C07303=1117.265,17.086,-52.064,179.768,6.707,149.300
C07304=1117.260,17.335,-52.079,179.769,6.711,149.301
C07305=1117.255,17.584,-52.094,179.769,6.716,149.302
C07306=1117.250,17.834,-52.108,179.770,6.720,149.303
C07307=1117.245,18.084,-52.123,179.771,6.725,149.303
C07308=1117.240,18.333,-52.138,179.772,6.729,149.304
C07309=1117.235,18.583,-52.152,179.773,6.734,149.305
C07310=1117.230,18.832,-52.168,179.774,6.738,149.306
C07311=1117.225,19.082,-52.182,179.774,6.742,149.306
C07312=1117.220,19.332,-52.196,179.775,6.747,149.307
C07313=1117.215,19.581,-52.211,179.776,6.751,149.308
C07314=1117.210,19.831,-52.226,179.776,6.756,149.309
C07315=1117.205,20.080,-52.241,179.777,6.760,149.309
C07316=1117.200,20.330,-52.255,179.778,6.764,149.310
C07317=1117.195,20.579,-52.271,179.779,6.769,149.311
C07318=1117.190,20.829,-52.285,179.780,6.773,149.312
C07319=1117.185,21.078,-52.300,179.781,6.778,149.312
C07320=1117.179,21.328,-52.315,179.782,6.782,149.313
C07321=1117.175,21.577,-52.330,179.783,6.787,149.314
C07322=1117.170,21.827,-52.344,179.783,6.791,149.315
C07323=1117.164,22.076,-52.360,179.784,6.796,149.315
C07324=1117.160,22.291,-52.372,179.785,6.799,149.316
C07325=1117.155,22.505,-52.385,179.785,6.803,149.317
C07326=1117.151,22.720,-52.397,179.786,6.807,149.317
C07327=1117.147,22.935,-52.410,179.787,6.810,149.318
C07328=1117.142,23.149,-52.424,179.787,6.814,149.318
C07329=1117.139,23.364,-52.436,179.788,6.818,149.319
C07330=1117.134,23.579,-52.449,179.789,6.822,149.320
C07331=1117.130,23.793,-52.462,179.790,6.826,149.320
C07332=1117.125,24.043,-52.477,179.790,6.829,149.321
C07333=1117.120,24.292,-52.492,179.791,6.834,149.322
C07334=1117.114,24.542,-52.507,179.792,6.838,149.322
C07335=1117.110,24.791,-52.522,179.793,6.843,149.323
C07336=1117.105,25.041,-52.537,179.794,6.847,149.324
C07337=1117.099,25.290,-52.552,179.795,6.851,149.324
C07338=1117.095,25.539,-52.567,179.796,6.856,149.325
C07339=1117.089,25.789,-52.582,179.797,6.860,149.326
C07340=1117.084,26.038,-52.597,179.798,6.865,149.327
C07341=1117.079,26.288,-52.613,179.799,6.869,149.327
C07342=1117.074,26.537,-52.628,179.800,6.873,149.328
C07343=1117.069,26.787,-52.643,179.800,6.877,149.329
C07344=1117.065,27.036,-52.658,179.801,6.882,149.329
C07345=1117.059,27.286,-52.673,179.802,6.886,149.330
C07346=1117.054,27.536,-52.688,179.803,6.890,149.331
C07347=1117.049,27.785,-52.703,179.804,6.895,149.331
C07348=1117.044,28.034,-52.718,179.805,6.899,149.332
C07349=1117.039,28.283,-52.734,179.806,6.904,149.333
C07350=1117.034,28.533,-52.749,179.807,6.908,149.334
C07351=1117.029,28.783,-52.764,179.808,6.912,149.334
C07352=1117.025,29.032,-52.779,179.809,6.917,149.335
C07353=1117.019,29.282,-52.795,179.809,6.920,149.336
C07354=1117.014,29.531,-52.810,179.810,6.924,149.336
C07355=1117.009,29.780,-52.825,179.812,6.929,149.337
C07356=1117.004,30.030,-52.841,179.813,6.933,149.337
C07357=1116.999,30.280,-52.855,179.814,6.937,149.338
C07358=1116.994,30.529,-52.871,179.815,6.942,149.339
C07359=1116.989,30.779,-52.886,179.815,6.946,149.340
C07360=1116.984,31.028,-52.902,179.816,6.951,149.340
C07361=1116.979,31.277,-52.917,179.817,6.955,149.341
C07362=1116.974,31.527,-52.933,179.818,6.958,149.342
C07363=1116.969,31.777,-52.948,179.819,6.963,149.342
C07364=1116.964,32.026,-52.963,179.820,6.967,149.343
C07365=1116.959,32.275,-52.979,179.821,6.971,149.344
C07366=1116.954,32.524,-52.994,179.822,6.976,149.344
C07367=1116.950,32.774,-53.010,179.823,6.980,149.345
C07368=1116.944,33.024,-53.025,179.824,6.984,149.346
C07369=1116.939,33.273,-53.041,179.825,6.989,149.346
C07370=1116.934,33.522,-53.056,179.826,6.993,149.347
C07371=1116.929,33.772,-53.072,179.827,6.996,149.347
C07372=1116.924,34.022,-53.087,179.828,7.001,149.348
C07373=1116.919,34.271,-53.102,179.829,7.005,149.349
C07374=1116.914,34.520,-53.118,179.830,7.009,149.349
C07375=1116.909,34.770,-53.134,179.831,7.014,149.350
C07376=1116.905,35.019,-53.149,179.832,7.018,149.351
C07377=1116.899,35.269,-53.164,179.833,7.022,149.351
C07378=1116.894,35.518,-53.180,179.834,7.027,149.352
C07379=1116.889,35.768,-53.196,179.835,7.031,149.353
C07380=1116.885,35.983,-53.210,179.836,7.034,149.353
C07381=1116.881,36.197,-53.222,179.837,7.038,149.354
C07382=1116.877,36.412,-53.236,179.838,7.041,149.354
C07383=1116.872,36.626,-53.250,179.839,7.045,149.355
C07384=1116.868,36.841,-53.263,179.840,7.048,149.355
C07385=1116.863,37.055,-53.276,179.841,7.052,149.356
C07386=1116.859,37.269,-53.290,179.842,7.056,149.356
C07387=1116.855,37.484,-53.304,179.842,7.059,149.357
C07388=1116.849,37.733,-53.319,179.843,7.063,149.358
C07389=1116.845,37.983,-53.335,179.845,7.067,149.358
C07390=1116.840,38.232,-53.350,179.846,7.072,149.359
C07391=1116.835,38.482,-53.366,179.847,7.076,149.359
C07392=1116.830,38.732,-53.382,179.848,7.080,149.360
C07393=1116.825,38.981,-53.398,179.848,7.084,149.361
C07394=1116.819,39.230,-53.414,179.849,7.088,149.361
C07395=1116.815,39.480,-53.430,179.850,7.092,149.362
C07396=1116.810,39.729,-53.445,179.852,7.096,149.362
C07397=1116.805,39.978,-53.461,179.853,7.101,149.363
C07398=1116.800,40.228,-53.477,179.854,7.105,149.364
C07399=1116.795,40.478,-53.492,179.855,7.109,149.364
C07400=1116.789,40.727,-53.508,179.856,7.114,149.365
C07401=1116.785,40.976,-53.525,179.857,7.117,149.366
C07402=1116.779,41.226,-53.540,179.858,7.121,149.366
C07403=1116.775,41.476,-53.556,179.859,7.125,149.367
C07404=1116.770,41.724,-53.572,179.860,7.130,149.367
C07405=1116.765,41.974,-53.588,179.861,7.134,149.368
C07406=1116.760,42.224,-53.603,179.863,7.138,149.369
C07407=1116.755,42.473,-53.620,179.864,7.142,149.369
C07408=1116.750,42.723,-53.636,179.865,7.146,149.370
C07409=1116.745,42.972,-53.651,179.866,7.150,149.370
C07410=1116.740,43.221,-53.668,179.867,7.154,149.371
C07411=1116.735,43.471,-53.684,179.868,7.158,149.372
C07412=1116.730,43.720,-53.700,179.869,7.162,149.372
C07413=1116.725,43.970,-53.716,179.870,7.167,149.373
C07414=1116.720,44.219,-53.731,179.871,7.171,149.374
C07415=1116.715,44.469,-53.748,179.873,7.175,149.374
C07416=1116.710,44.718,-53.764,179.873,7.178,149.375
C07417=1116.705,44.967,-53.780,179.875,7.183,149.375
C07418=1116.700,45.217,-53.796,179.876,7.187,149.376
C07419=1116.695,45.466,-53.812,179.877,7.191,149.376
C07420=1116.690,45.716,-53.828,179.878,7.195,149.377
C07421=1116.685,45.965,-53.844,179.879,7.200,149.378
C07422=1116.680,46.215,-53.860,179.881,7.204,149.378
C07423=1116.675,46.464,-53.877,179.882,7.208,149.379
C07424=1116.670,46.714,-53.893,179.882,7.211,149.379
C07425=1116.665,46.963,-53.909,179.884,7.215,149.380
C07426=1116.660,47.213,-53.925,179.885,7.220,149.380
C07427=1116.655,47.461,-53.941,179.886,7.224,149.381
C07428=1116.651,47.711,-53.958,179.888,7.228,149.382
C07429=1116.646,47.960,-53.974,179.889,7.232,149.382
C07430=1116.641,48.210,-53.990,179.890,7.236,149.383
C07431=1116.636,48.459,-54.006,179.891,7.240,149.383
C07432=1116.631,48.709,-54.022,179.892,7.244,149.384
C07433=1116.626,48.958,-54.039,179.893,7.248,149.384
C07434=1116.621,49.208,-54.055,179.895,7.252,149.385
C07435=1116.616,49.457,-54.072,179.896,7.256,149.386
C07436=1116.610,49.781,-54.093,179.897,7.261,149.386
C07437=1116.603,50.104,-54.114,179.899,7.267,149.387
C07438=1116.597,50.427,-54.135,179.900,7.272,149.388
C07439=1116.591,50.750,-54.156,179.902,7.277,149.388
C07440=1116.585,51.000,-54.173,179.903,7.281,149.389
C07441=1116.580,51.249,-54.190,179.905,7.285,149.390
C07442=1116.576,51.499,-54.206,179.906,7.290,149.390
C07443=1116.571,51.748,-54.222,179.906,7.293,149.391
C07444=1116.566,51.997,-54.239,179.908,7.297,149.391
C07445=1116.560,52.247,-54.255,179.909,7.301,149.392
C07446=1116.556,52.497,-54.271,179.910,7.305,149.392
C07447=1116.550,52.745,-54.288,179.911,7.309,149.393
C07448=1116.546,52.995,-54.304,179.913,7.313,149.393
C07449=1116.541,53.245,-54.322,179.914,7.318,149.394
C07450=1116.536,53.493,-54.338,179.915,7.322,149.395
C07451=1116.531,53.744,-54.354,179.916,7.325,149.395
C07452=1116.526,53.993,-54.371,179.917,7.329,149.396
C07453=1116.521,54.242,-54.387,179.919,7.333,149.396
C07454=1116.516,54.492,-54.404,179.920,7.338,149.397
C07455=1116.511,54.740,-54.420,179.921,7.342,149.397
C07456=1116.507,54.990,-54.437,179.923,7.346,149.398
C07457=1116.501,55.240,-54.454,179.924,7.350,149.398
C07458=1116.496,55.489,-54.470,179.925,7.354,149.399
C07459=1116.491,55.739,-54.487,179.926,7.357,149.399
C07460=1116.486,55.988,-54.504,179.927,7.361,149.400
C07461=1116.481,56.237,-54.520,179.929,7.365,149.401
C07462=1116.477,56.487,-54.537,179.930,7.370,149.401
C07463=1116.471,56.736,-54.554,179.931,7.374,149.402
C07464=1116.465,57.091,-54.578,179.933,7.379,149.402
C07465=1116.458,57.446,-54.601,179.935,7.385,149.403
C07466=1116.450,57.801,-54.626,179.937,7.391,149.404
C07467=1116.444,58.155,-54.649,179.939,7.396,149.405
C07468=1116.438,58.405,-54.666,179.940,7.401,149.405
C07469=1116.434,58.655,-54.683,179.941,7.404,149.406
C07470=1116.429,58.903,-54.699,179.942,7.409,149.406
C07471=1116.424,59.153,-54.716,179.944,7.413,149.407
C07472=1116.419,59.403,-54.733,179.944,7.416,149.407
C07473=1116.414,59.652,-54.750,179.946,7.420,149.408
C07474=1116.409,59.901,-54.767,179.947,7.424,149.409
C07475=1116.404,60.151,-54.784,179.949,7.428,149.409
C07476=1116.399,60.400,-54.801,179.950,7.432,149.409
C07477=1116.394,60.649,-54.818,179.951,7.436,149.410
C07478=1116.389,60.898,-54.835,179.953,7.440,149.410
C07479=1116.385,61.148,-54.852,179.954,7.445,149.411
C07480=1116.379,61.398,-54.869,179.955,7.449,149.412
C07481=1116.375,61.647,-54.886,179.956,7.452,149.412
C07482=1116.369,61.896,-54.902,179.958,7.456,149.413
C07483=1116.365,62.145,-54.920,179.959,7.460,149.413
C07484=1116.360,62.395,-54.937,179.960,7.464,149.414
C07485=1116.355,62.644,-54.954,179.962,7.468,149.414
C07486=1116.350,62.894,-54.971,179.963,7.472,149.415
C07487=1116.345,63.143,-54.987,179.964,7.476,149.415
C07488=1116.341,63.358,-55.003,179.965,7.479,149.416
C07489=1116.337,63.571,-55.017,179.966,7.483,149.416
C07490=1116.333,63.786,-55.033,179.968,7.486,149.417
C07491=1116.328,64.001,-55.046,179.969,7.490,149.417
C07492=1116.324,64.215,-55.061,179.970,7.493,149.417
C07493=1116.320,64.429,-55.076,179.971,7.497,149.418
C07494=1116.316,64.643,-55.091,179.972,7.500,149.418
C07495=1116.311,64.858,-55.106,179.974,7.504,149.419
C07496=1116.307,65.107,-55.123,179.974,7.507,149.419
C07497=1116.301,65.356,-55.140,179.976,7.511,149.420
C07498=1116.297,65.606,-55.157,179.977,7.515,149.420
C07499=1116.292,65.855,-55.175,179.979,7.519,149.421
C07500=1116.287,66.104,-55.191,179.980,7.523,149.421
C07501=1116.282,66.354,-55.209,179.982,7.527,149.422
C07502=1116.277,66.603,-55.227,179.983,7.531,149.422
C07503=1116.273,66.853,-55.243,179.984,7.535,149.423
C07504=1116.267,67.102,-55.260,179.986,7.540,149.423
C07505=1116.262,67.351,-55.278,179.987,7.543,149.424
C07506=1116.258,67.601,-55.295,179.988,7.547,149.424
C07507=1116.253,67.850,-55.313,179.989,7.551,149.425
C07508=1116.247,68.100,-55.330,179.991,7.555,149.425
C07509=1116.243,68.348,-55.347,179.992,7.559,149.426
C07510=1116.238,68.598,-55.365,179.993,7.563,149.426
C07511=1116.233,68.847,-55.383,179.995,7.567,149.427
C07512=1116.229,69.097,-55.399,179.997,7.571,149.427
C07513=1116.224,69.346,-55.417,179.998,7.575,149.428
C07514=1116.218,69.596,-55.435,179.999,7.579,149.428
C07515=1116.214,69.844,-55.452,-179.999,7.583,149.429
C07516=1116.208,70.094,-55.469,-179.998,7.587,149.429
C07517=1116.204,70.343,-55.487,-179.997,7.590,149.430
C07518=1116.198,70.593,-55.504,-179.996,7.594,149.430
C07519=1116.194,70.842,-55.521,-179.994,7.598,149.431
C07520=1116.189,71.091,-55.539,-179.993,7.602,149.431
C07521=1116.184,71.341,-55.557,-179.991,7.606,149.432
C07522=1116.179,71.590,-55.574,-179.990,7.610,149.432
C07523=1116.175,71.839,-55.591,-179.989,7.614,149.433
C07524=1116.170,72.088,-55.609,-179.987,7.618,149.433
C07525=1116.165,72.338,-55.627,-179.985,7.622,149.434
C07526=1116.160,72.587,-55.645,-179.984,7.626,149.434
C07527=1116.155,72.837,-55.663,-179.983,7.630,149.435
C07528=1116.150,73.086,-55.679,-179.981,7.634,149.435
C07529=1116.145,73.335,-55.697,-179.980,7.638,149.436
C07530=1116.140,73.585,-55.714,-179.979,7.642,149.436
C07531=1116.135,73.834,-55.732,-179.978,7.646,149.437
C07532=1116.130,74.083,-55.750,-179.976,7.650,149.437
C07533=1116.125,74.333,-55.768,-179.974,7.653,149.438
C07534=1116.121,74.582,-55.785,-179.973,7.658,149.438
C07535=1116.116,74.831,-55.803,-179.972,7.662,149.439
C07536=1116.111,75.080,-55.821,-179.970,7.666,149.439
C07537=1116.106,75.330,-55.839,-179.969,7.669,149.440
C07538=1116.101,75.579,-55.856,-179.967,7.674,149.440
C07539=1116.096,75.829,-55.874,-179.966,7.678,149.441
C07540=1116.091,76.078,-55.892,-179.964,7.681,149.441
C07541=1116.086,76.327,-55.910,-179.963,7.685,149.442
C07542=1116.082,76.577,-55.928,-179.962,7.690,149.442
C07543=1116.077,76.827,-55.946,-179.960,7.694,149.443
C07544=1116.073,77.040,-55.961,-179.959,7.697,149.443
C07545=1116.069,77.254,-55.976,-179.958,7.700,149.444
C07546=1116.064,77.468,-55.991,-179.958,7.703,149.444
C07547=1116.060,77.683,-56.007,-179.957,7.706,149.445
C07548=1116.056,77.897,-56.023,-179.956,7.709,149.445
C07549=1116.051,78.111,-56.038,-179.955,7.712,149.445
C07550=1116.047,78.326,-56.053,-179.954,7.715,149.446
C07551=1116.043,78.541,-56.069,-179.954,7.718,149.447
C07552=1116.038,78.790,-56.087,-179.952,7.722,149.447
C07553=1116.033,79.039,-56.105,-179.952,7.726,149.448
C07554=1116.028,79.288,-56.123,-179.950,7.730,149.448
C07555=1116.024,79.537,-56.141,-179.950,7.733,149.449
C07556=1116.019,79.787,-56.159,-179.948,7.737,149.449
C07557=1116.014,80.036,-56.177,-179.948,7.741,149.450
C07558=1116.009,80.285,-56.195,-179.946,7.745,149.450
C07559=1116.004,80.534,-56.213,-179.945,7.748,149.451
C07560=1116.000,80.784,-56.231,-179.944,7.752,149.451
C07561=1115.995,81.033,-56.249,-179.943,7.756,149.452
C07562=1115.990,81.282,-56.267,-179.942,7.760,149.453
C07563=1115.985,81.532,-56.285,-179.941,7.764,149.453
C07564=1115.980,81.781,-56.303,-179.940,7.767,149.453
C07565=1115.975,82.030,-56.321,-179.939,7.771,149.454
C07566=1115.971,82.280,-56.339,-179.938,7.774,149.454
C07567=1115.966,82.529,-56.357,-179.936,7.778,149.455
C07568=1115.961,82.778,-56.375,-179.935,7.782,149.456
C07569=1115.956,83.027,-56.393,-179.934,7.786,149.456
C07570=1115.951,83.276,-56.411,-179.933,7.790,149.457
C07571=1115.946,83.526,-56.429,-179.932,7.794,149.457
C07572=1115.942,83.776,-56.447,-179.931,7.797,149.458
C07573=1115.936,84.025,-56.466,-179.930,7.801,149.458
C07574=1115.931,84.274,-56.484,-179.929,7.804,149.459
C07575=1115.926,84.523,-56.502,-179.927,7.808,149.459
C07576=1115.922,84.772,-56.521,-179.926,7.813,149.460
C07577=1115.917,85.022,-56.539,-179.925,7.816,149.460
C07578=1115.913,85.271,-56.557,-179.924,7.820,149.461
C07579=1115.908,85.520,-56.575,-179.922,7.824,149.461
C07580=1115.902,85.770,-56.593,-179.921,7.827,149.462
C07581=1115.898,86.020,-56.612,-179.920,7.831,149.462
C07582=1115.893,86.269,-56.630,-179.919,7.835,149.463
C07583=1115.888,86.517,-56.648,-179.917,7.840,149.464
C07584=1115.883,86.766,-56.666,-179.916,7.843,149.464
C07585=1115.878,87.016,-56.684,-179.915,7.847,149.464
C07586=1115.873,87.266,-56.703,-179.914,7.851,149.465
C07587=1115.869,87.514,-56.722,-179.913,7.854,149.465
C07588=1115.864,87.764,-56.740,-179.911,7.858,149.466
C07589=1115.859,88.013,-56.758,-179.910,7.862,149.467
C07590=1115.854,88.263,-56.777,-179.908,7.866,149.467
C07591=1115.849,88.511,-56.796,-179.907,7.870,149.467
C07592=1115.844,88.761,-56.814,-179.906,7.873,149.468
C07593=1115.840,89.010,-56.832,-179.905,7.877,149.469
C07594=1115.834,89.260,-56.851,-179.903,7.881,149.469
C07595=1115.830,89.509,-56.869,-179.901,7.885,149.469
C07596=1115.825,89.758,-56.887,-179.901,7.888,149.470
C07597=1115.820,90.008,-56.906,-179.899,7.892,149.470
C07598=1115.815,90.256,-56.925,-179.898,7.896,149.471
C07599=1115.810,90.506,-56.943,-179.896,7.900,149.471
C07600=1115.806,90.720,-56.959,-179.895,7.903,149.472
C07601=1115.803,90.934,-56.975,-179.894,7.906,149.472
C07602=1115.798,91.149,-56.990,-179.893,7.910,149.473
C07603=1115.794,91.363,-57.007,-179.892,7.913,149.473
C07604=1115.789,91.576,-57.023,-179.891,7.917,149.473
C07605=1115.786,91.790,-57.039,-179.889,7.920,149.474
C07606=1115.782,92.005,-57.055,-179.888,7.923,149.474
C07607=1115.778,92.219,-57.070,-179.887,7.926,149.475
C07608=1115.772,92.468,-57.090,-179.885,7.930,149.475
C07609=1115.767,92.717,-57.108,-179.884,7.934,149.475
C07610=1115.763,92.967,-57.127,-179.882,7.938,149.476
C07611=1115.758,93.216,-57.145,-179.881,7.942,149.476
C07612=1115.754,93.465,-57.164,-179.879,7.946,149.477
C07613=1115.748,93.715,-57.183,-179.878,7.950,149.477
C07614=1115.744,93.963,-57.202,-179.877,7.953,149.478
C07615=1115.738,94.214,-57.221,-179.875,7.957,149.478
C07616=1115.734,94.462,-57.239,-179.873,7.961,149.479
C07617=1115.729,94.711,-57.257,-179.872,7.965,149.479
C07618=1115.724,94.961,-57.277,-179.870,7.969,149.480
C07619=1115.719,95.210,-57.295,-179.869,7.973,149.480
C07620=1115.715,95.460,-57.315,-179.867,7.976,149.480
C07621=1115.710,95.708,-57.333,-179.865,7.980,149.481
C07622=1115.705,95.958,-57.352,-179.864,7.984,149.481
C07623=1115.700,96.207,-57.371,-179.862,7.988,149.482
C07624=1115.695,96.456,-57.390,-179.861,7.992,149.482
C07625=1115.691,96.706,-57.409,-179.859,7.996,149.483
C07626=1115.685,96.954,-57.428,-179.857,8.000,149.483
C07627=1115.681,97.204,-57.446,-179.856,8.004,149.483
C07628=1115.676,97.453,-57.465,-179.854,8.008,149.484
C07629=1115.672,97.703,-57.485,-179.853,8.011,149.484
C07630=1115.666,97.952,-57.503,-179.851,8.015,149.485
C07631=1115.662,98.201,-57.522,-179.849,8.019,149.485
C07632=1115.657,98.450,-57.541,-179.847,8.023,149.485
C07633=1115.652,98.699,-57.559,-179.846,8.027,149.486
C07634=1115.647,98.949,-57.579,-179.844,8.030,149.486
C07635=1115.642,99.197,-57.598,-179.843,8.034,149.487
C07636=1115.638,99.447,-57.617,-179.841,8.038,149.487
C07637=1115.633,99.696,-57.635,-179.839,8.042,149.487
C07638=1115.628,99.946,-57.655,-179.837,8.046,149.488
C07639=1115.623,100.195,-57.674,-179.836,8.050,149.488
C07640=1115.619,100.444,-57.693,-179.834,8.053,149.489
C07641=1115.613,100.693,-57.713,-179.832,8.057,149.489
C07642=1115.609,100.943,-57.731,-179.830,8.061,149.489
C07643=1115.604,101.192,-57.751,-179.829,8.065,149.490
C07644=1115.599,101.441,-57.770,-179.827,8.068,149.490
C07645=1115.595,101.690,-57.789,-179.825,8.072,149.490
C07646=1115.590,101.939,-57.808,-179.824,8.076,149.491
C07647=1115.585,102.189,-57.828,-179.822,8.079,149.491
C07648=1115.580,102.437,-57.847,-179.820,8.083,149.491
C07649=1115.575,102.687,-57.866,-179.818,8.087,149.492
C07650=1115.570,102.936,-57.886,-179.816,8.091,149.492
C07651=1115.566,103.186,-57.904,-179.814,8.095,149.493
C07652=1115.560,103.434,-57.923,-179.812,8.099,149.493
C07653=1115.556,103.684,-57.943,-179.810,8.103,149.493
C07654=1115.552,103.933,-57.962,-179.809,8.107,149.494
C07655=1115.546,104.182,-57.981,-179.807,8.110,149.494
C07656=1115.542,104.396,-57.999,-179.806,8.113,149.494
C07657=1115.538,104.610,-58.015,-179.804,8.117,149.495
C07658=1115.534,104.824,-58.032,-179.802,8.120,149.495
C07659=1115.530,105.038,-58.048,-179.800,8.123,149.495
C07660=1115.526,105.252,-58.065,-179.799,8.127,149.495
C07661=1115.522,105.466,-58.081,-179.797,8.130,149.496
C07662=1115.518,105.680,-58.099,-179.795,8.133,149.496
C07663=1115.514,105.894,-58.115,-179.794,8.136,149.496
C07664=1115.509,106.144,-58.134,-179.792,8.140,149.496
C07665=1115.504,106.393,-58.154,-179.789,8.144,149.497
C07666=1115.499,106.642,-58.173,-179.788,8.148,149.497
C07667=1115.494,106.892,-58.193,-179.786,8.151,149.497
C07668=1115.490,107.140,-58.212,-179.784,8.155,149.498
C07669=1115.485,107.389,-58.232,-179.782,8.159,149.498
C07670=1115.480,107.639,-58.252,-179.780,8.162,149.498
C07671=1115.475,107.888,-58.271,-179.777,8.167,149.498
C07672=1115.470,108.137,-58.291,-179.776,8.170,149.499
C07673=1115.466,108.387,-58.310,-179.774,8.174,149.499
C07674=1115.461,108.636,-58.331,-179.772,8.177,149.499
C07675=1115.457,108.884,-58.349,-179.770,8.181,149.500
C07676=1115.452,109.134,-58.369,-179.767,8.186,149.500
C07677=1115.447,109.384,-58.389,-179.765,8.189,149.500
C07678=1115.442,109.632,-58.409,-179.763,8.193,149.500
C07679=1115.437,109.881,-58.428,-179.761,8.196,149.501
C07680=1115.433,110.131,-58.448,-179.759,8.200,149.501
C07681=1115.427,110.380,-58.467,-179.756,8.204,149.501
C07682=1115.423,110.629,-58.488,-179.754,8.207,149.501
C07683=1115.418,110.878,-58.507,-179.753,8.211,149.502
C07684=1115.413,111.128,-58.527,-179.751,8.215,149.502
C07685=1115.408,111.376,-58.547,-179.749,8.218,149.502
C07686=1115.403,111.626,-58.567,-179.747,8.222,149.502
C07687=1115.399,111.875,-58.586,-179.746,8.225,149.503
C07688=1115.394,112.124,-58.607,-179.743,8.228,149.503
C07689=1115.389,112.373,-58.626,-179.741,8.232,149.503
C07690=1115.385,112.622,-58.646,-179.740,8.236,149.504
C07691=1115.380,112.872,-58.666,-179.738,8.239,149.504
C07692=1115.375,113.121,-58.686,-179.736,8.243,149.504
C07693=1115.371,113.370,-58.706,-179.735,8.246,149.505
C07694=1115.365,113.619,-58.725,-179.733,8.249,149.505
C07695=1115.361,113.868,-58.746,-179.731,8.253,149.505
C07696=1115.356,114.118,-58.765,-179.728,8.256,149.505
C07697=1115.352,114.367,-58.786,-179.728,8.259,149.506
C07698=1115.347,114.616,-58.805,-179.725,8.263,149.506
C07699=1115.342,114.864,-58.825,-179.723,8.266,149.506
C07700=1115.337,115.114,-58.845,-179.722,8.270,149.507
C07701=1115.333,115.363,-58.865,-179.720,8.274,149.507
C07702=1115.327,115.613,-58.886,-179.718,8.277,149.507
C07703=1115.323,115.862,-58.906,-179.716,8.280,149.507
C07704=1115.318,116.111,-58.926,-179.715,8.284,149.508
C07705=1115.313,116.359,-58.946,-179.713,8.287,149.508
C07706=1115.308,116.609,-58.965,-179.711,8.290,149.508
C07707=1115.304,116.858,-58.986,-179.709,8.294,149.508
C07708=1115.299,117.107,-59.006,-179.707,8.298,149.509
C07709=1115.295,117.357,-59.026,-179.705,8.301,149.509
C07710=1115.289,117.606,-59.047,-179.704,8.304,149.509
C07711=1115.285,117.855,-59.066,-179.702,8.308,149.510
C07712=1115.280,118.069,-59.084,-179.701,8.310,149.510
C07713=1115.277,118.283,-59.101,-179.699,8.314,149.510
C07714=1115.273,118.496,-59.118,-179.697,8.317,149.510
C07715=1115.268,118.710,-59.135,-179.696,8.319,149.511
C07716=1115.265,118.925,-59.153,-179.694,8.322,149.511
C07717=1115.261,119.138,-59.171,-179.693,8.325,149.511
C07718=1115.256,119.352,-59.188,-179.691,8.328,149.511
C07719=1115.252,119.566,-59.205,-179.690,8.331,149.512
C07720=1115.248,119.815,-59.226,-179.687,8.334,149.512
C07721=1115.243,120.065,-59.245,-179.686,8.338,149.512
C07722=1115.238,120.314,-59.266,-179.684,8.341,149.512
C07723=1115.233,120.563,-59.287,-179.682,8.345,149.513
C07724=1115.229,120.812,-59.307,-179.680,8.348,149.513
C07725=1115.224,121.061,-59.327,-179.679,8.351,149.513
C07726=1115.219,121.311,-59.348,-179.677,8.355,149.514
C07727=1115.214,121.560,-59.368,-179.675,8.358,149.514
C07728=1115.210,121.808,-59.388,-179.674,8.361,149.514
C07729=1115.206,122.057,-59.409,-179.672,8.364,149.514
C07730=1115.200,122.307,-59.429,-179.670,8.368,149.515
C07731=1115.196,122.556,-59.449,-179.668,8.372,149.515
C07732=1115.191,122.805,-59.470,-179.667,8.374,149.515
C07733=1115.186,123.054,-59.491,-179.664,8.378,149.515
C07734=1115.182,123.303,-59.511,-179.663,8.382,149.516
C07735=1115.177,123.552,-59.532,-179.661,8.385,149.516
C07736=1115.172,123.802,-59.553,-179.659,8.388,149.516
C07737=1115.168,124.051,-59.573,-179.657,8.392,149.516
C07738=1115.163,124.300,-59.593,-179.656,8.395,149.517
C07739=1115.158,124.549,-59.613,-179.654,8.398,149.517
C07740=1115.153,124.798,-59.634,-179.652,8.402,149.517
C07741=1115.149,125.047,-59.654,-179.650,8.405,149.518
C07742=1115.144,125.297,-59.675,-179.649,8.408,149.518
C07743=1115.139,125.545,-59.696,-179.647,8.412,149.518
C07744=1115.134,125.795,-59.717,-179.645,8.415,149.518
C07745=1115.130,126.044,-59.737,-179.644,8.418,149.519
C07746=1115.125,126.293,-59.757,-179.641,8.421,149.519
C07747=1115.120,126.542,-59.778,-179.640,8.425,149.519
C07748=1115.115,126.791,-59.799,-179.638,8.428,149.520
C07749=1115.110,127.040,-59.820,-179.636,8.432,149.520
C07750=1115.106,127.289,-59.840,-179.634,8.435,149.520
C07751=1115.101,127.538,-59.862,-179.633,8.438,149.520
C07752=1115.097,127.787,-59.882,-179.631,8.442,149.521
C07753=1115.092,128.036,-59.902,-179.629,8.445,149.521
C07754=1115.087,128.285,-59.923,-179.628,8.448,149.521
C07755=1115.083,128.534,-59.944,-179.626,8.452,149.522
C07756=1115.078,128.784,-59.965,-179.624,8.455,149.522
C07757=1115.074,129.033,-59.985,-179.623,8.458,149.522
C07758=1115.068,129.282,-60.006,-179.620,8.461,149.522
C07759=1115.063,129.531,-60.027,-179.619,8.465,149.523
C07760=1115.059,129.780,-60.048,-179.617,8.468,149.523
C07761=1115.054,130.029,-60.069,-179.615,8.471,149.523
C07762=1115.049,130.278,-60.090,-179.613,8.475,149.523
C07763=1115.044,130.527,-60.111,-179.612,8.478,149.524
C07764=1115.040,130.776,-60.131,-179.610,8.482,149.524
C07765=1115.035,131.025,-60.153,-179.608,8.485,149.524
C07766=1115.031,131.274,-60.174,-179.607,8.488,149.525
C07767=1115.026,131.524,-60.195,-179.605,8.492,149.525
C07768=1115.022,131.737,-60.212,-179.604,8.494,149.525
C07769=1115.018,131.951,-60.230,-179.602,8.497,149.525
C07770=1115.013,132.165,-60.248,-179.601,8.500,149.526
C07771=1115.009,132.378,-60.267,-179.599,8.503,149.526
C07772=1115.006,132.593,-60.284,-179.597,8.506,149.526
C07773=1115.002,132.806,-60.302,-179.596,8.509,149.526
C07774=1114.997,133.021,-60.321,-179.595,8.512,149.527
C07775=1114.993,133.234,-60.339,-179.593,8.515,149.527
C07776=1114.989,133.483,-60.359,-179.591,8.518,149.527
C07777=1114.984,133.732,-60.380,-179.590,8.521,149.527
C07778=1114.979,133.981,-60.402,-179.588,8.525,149.528
C07779=1114.975,134.231,-60.423,-179.586,8.528,149.528
C07780=1114.970,134.479,-60.444,-179.585,8.531,149.528
C07781=1114.965,134.728,-60.465,-179.583,8.535,149.529
C07782=1114.961,134.977,-60.486,-179.581,8.538,149.529
C07783=1114.956,135.226,-60.507,-179.580,8.541,149.529
C07784=1114.951,135.476,-60.529,-179.578,8.545,149.530
C07785=1114.947,135.724,-60.550,-179.576,8.548,149.530
C07786=1114.942,135.974,-60.571,-179.574,8.551,149.530
C07787=1114.937,136.223,-60.592,-179.573,8.555,149.531
C07788=1114.932,136.472,-60.614,-179.571,8.558,149.531
C07789=1114.928,136.721,-60.634,-179.569,8.561,149.531
C07790=1114.923,136.970,-60.656,-179.568,8.565,149.531
C07791=1114.918,137.219,-60.677,-179.566,8.568,149.532
C07792=1114.914,137.468,-60.698,-179.564,8.571,149.532
C07793=1114.909,137.717,-60.719,-179.562,8.575,149.532
C07794=1114.904,137.966,-60.741,-179.561,8.578,149.533
C07795=1114.899,138.215,-60.762,-179.559,8.581,149.533
C07796=1114.895,138.465,-60.784,-179.557,8.585,149.533
C07797=1114.891,138.714,-60.804,-179.556,8.588,149.534
C07798=1114.886,138.962,-60.826,-179.554,8.592,149.534
C07799=1114.881,139.212,-60.848,-179.552,8.595,149.534
C07800=1114.876,139.461,-60.869,-179.551,8.598,149.534
C07801=1114.871,139.709,-60.891,-179.549,8.602,149.535
C07802=1114.867,139.958,-60.911,-179.547,8.605,149.535
C07803=1114.863,140.208,-60.933,-179.546,8.608,149.536
C07804=1114.858,140.456,-60.955,-179.544,8.612,149.536
C07805=1114.853,140.706,-60.976,-179.543,8.615,149.536
C07806=1114.848,140.955,-60.998,-179.541,8.618,149.536
C07807=1114.844,141.203,-61.019,-179.539,8.622,149.537
C07808=1114.839,141.453,-61.040,-179.538,8.625,149.537
C07809=1114.835,141.702,-61.062,-179.536,8.628,149.537
C07810=1114.830,141.951,-61.084,-179.534,8.632,149.538
C07811=1114.825,142.200,-61.105,-179.533,8.635,149.538
C07812=1114.820,142.449,-61.127,-179.531,8.639,149.538
C07813=1114.816,142.698,-61.148,-179.529,8.642,149.539
C07814=1114.811,142.947,-61.170,-179.528,8.645,149.539
C07815=1114.806,143.196,-61.191,-179.526,8.649,149.539
C07816=1114.802,143.445,-61.212,-179.525,8.652,149.540
C07817=1114.798,143.694,-61.234,-179.523,8.656,149.540
C07818=1114.793,143.943,-61.256,-179.521,8.659,149.540
C07819=1114.788,144.192,-61.277,-179.520,8.662,149.541
C07820=1114.783,144.441,-61.299,-179.518,8.666,149.541
C07821=1114.779,144.690,-61.321,-179.516,8.669,149.541
C07822=1114.774,144.939,-61.343,-179.515,8.673,149.542
C07823=1114.769,145.188,-61.365,-179.513,8.676,149.542
C07824=1114.765,145.402,-61.384,-179.511,8.680,149.542
C07825=1114.761,145.615,-61.402,-179.509,8.682,149.542
C07826=1114.757,145.829,-61.421,-179.507,8.686,149.543
C07827=1114.753,146.043,-61.439,-179.505,8.689,149.543
C07828=1114.749,146.257,-61.458,-179.504,8.692,149.543
C07829=1114.745,146.470,-61.476,-179.502,8.695,149.543
C07830=1114.741,146.684,-61.495,-179.500,8.698,149.544
C07831=1114.737,146.898,-61.514,-179.498,8.702,149.544
C07832=1114.732,147.147,-61.536,-179.496,8.705,149.544
C07833=1114.728,147.396,-61.558,-179.494,8.709,149.544
C07834=1114.723,147.645,-61.580,-179.491,8.713,149.545
C07835=1114.718,147.894,-61.601,-179.489,8.716,149.545
C07836=1114.714,148.143,-61.624,-179.487,8.720,149.545
C07837=1114.709,148.392,-61.645,-179.485,8.723,149.545
C07838=1114.705,148.641,-61.667,-179.483,8.727,149.546
C07839=1114.700,148.890,-61.689,-179.481,8.730,149.546
C07840=1114.696,149.139,-61.711,-179.479,8.734,149.546
C07841=1114.691,149.388,-61.733,-179.476,8.738,149.546
C07842=1114.686,149.637,-61.755,-179.474,8.742,149.546
C07843=1114.681,149.886,-61.777,-179.472,8.745,149.547
C07844=1114.677,150.135,-61.799,-179.470,8.749,149.547
C07845=1114.672,150.384,-61.821,-179.468,8.752,149.547
C07846=1114.668,150.633,-61.843,-179.466,8.755,149.547
C07847=1114.663,150.882,-61.864,-179.463,8.759,149.547
C07848=1114.658,151.131,-61.887,-179.461,8.762,149.548
C07849=1114.653,151.379,-61.909,-179.459,8.766,149.548
C07850=1114.649,151.629,-61.932,-179.456,8.770,149.548
C07851=1114.644,151.877,-61.953,-179.454,8.773,149.548
C07852=1114.640,152.127,-61.975,-179.452,8.777,149.549
C07853=1114.635,152.376,-61.998,-179.449,8.780,149.549
C07854=1114.630,152.625,-62.020,-179.447,8.783,149.549
C07855=1114.626,152.874,-62.042,-179.445,8.787,149.549
C07856=1114.621,153.122,-62.064,-179.443,8.790,149.549
C07857=1114.616,153.372,-62.087,-179.441,8.793,149.549
C07858=1114.611,153.621,-62.108,-179.439,8.797,149.550
C07859=1114.607,153.869,-62.131,-179.437,8.800,149.550
C07860=1114.603,154.119,-62.153,-179.434,8.804,149.550
C07861=1114.597,154.368,-62.175,-179.432,8.807,149.550
C07862=1114.593,154.616,-62.198,-179.430,8.811,149.550
C07863=1114.589,154.865,-62.220,-179.428,8.814,149.551
C07864=1114.584,155.115,-62.243,-179.425,8.817,149.551
C07865=1114.580,155.363,-62.265,-179.423,8.821,149.551
C07866=1114.575,155.612,-62.287,-179.421,8.824,149.551
C07867=1114.570,155.862,-62.310,-179.419,8.827,149.551
C07868=1114.566,156.110,-62.332,-179.416,8.831,149.551
C07869=1114.561,156.359,-62.354,-179.414,8.834,149.552
C07870=1114.556,156.608,-62.377,-179.412,8.837,149.552
C07871=1114.551,156.857,-62.399,-179.410,8.841,149.552
C07872=1114.547,157.106,-62.421,-179.408,8.844,149.552
C07873=1114.542,157.355,-62.445,-179.405,8.847,149.552
C07874=1114.537,157.604,-62.466,-179.404,8.850,149.552
C07875=1114.533,157.853,-62.489,-179.401,8.853,149.552
C07876=1114.528,158.102,-62.512,-179.399,8.857,149.553
C07877=1114.524,158.350,-62.534,-179.397,8.860,149.553
C07878=1114.519,158.600,-62.557,-179.395,8.863,149.553
C07879=1114.515,158.849,-62.579,-179.392,8.867,149.553
C07880=1114.511,159.063,-62.599,-179.391,8.869,149.553
C07881=1114.506,159.276,-62.618,-179.388,8.872,149.553
C07882=1114.503,159.489,-62.638,-179.387,8.875,149.553
C07883=1114.499,159.703,-62.657,-179.385,8.877,149.553
C07884=1114.495,159.917,-62.677,-179.383,8.881,149.554
C07885=1114.491,160.130,-62.696,-179.381,8.883,149.554
C07886=1114.487,160.345,-62.716,-179.379,8.886,149.554
C07887=1114.483,160.558,-62.735,-179.377,8.889,149.554
C07888=1114.478,160.807,-62.757,-179.375,8.892,149.554
C07889=1114.474,161.056,-62.780,-179.373,8.895,149.554
C07890=1114.470,161.305,-62.803,-179.371,8.898,149.555
C07891=1114.464,161.554,-62.825,-179.368,8.901,149.555
C07892=1114.460,161.802,-62.848,-179.366,8.904,149.555
C07893=1114.455,162.051,-62.872,-179.364,8.908,149.555
C07894=1114.451,162.301,-62.894,-179.361,8.911,149.555
C07895=1114.446,162.549,-62.917,-179.359,8.915,149.555
C07896=1114.442,162.798,-62.939,-179.357,8.917,149.555
C07897=1114.437,163.047,-62.963,-179.355,8.920,149.555
C07898=1114.433,163.296,-62.985,-179.352,8.923,149.555
C07899=1114.428,163.545,-63.008,-179.350,8.927,149.556
C07900=1114.423,163.793,-63.031,-179.348,8.930,149.556
C07901=1114.419,164.042,-63.054,-179.346,8.932,149.556
C07902=1114.414,164.292,-63.077,-179.344,8.936,149.556
C07903=1114.410,164.541,-63.099,-179.341,8.939,149.556
C07904=1114.405,164.790,-63.123,-179.339,8.942,149.556
C07905=1114.401,165.039,-63.146,-179.337,8.946,149.556
C07906=1114.396,165.287,-63.168,-179.335,8.948,149.556
C07907=1114.391,165.536,-63.192,-179.333,8.951,149.557
C07908=1114.386,165.785,-63.214,-179.330,8.954,149.557
C07909=1114.382,166.034,-63.237,-179.328,8.958,149.557
C07910=1114.378,166.283,-63.261,-179.326,8.961,149.557
C07911=1114.373,166.532,-63.284,-179.324,8.963,149.557
C07912=1114.368,166.780,-63.306,-179.322,8.967,149.557
C07913=1114.364,167.029,-63.330,-179.319,8.970,149.557
C07914=1114.359,167.278,-63.353,-179.317,8.973,149.557
C07915=1114.355,167.527,-63.376,-179.315,8.976,149.557
C07916=1114.350,167.776,-63.399,-179.313,8.979,149.557
C07917=1114.346,168.025,-63.422,-179.310,8.982,149.558
C07918=1114.341,168.274,-63.446,-179.308,8.986,149.558
C07919=1114.337,168.523,-63.469,-179.306,8.988,149.558
C07920=1114.332,168.771,-63.492,-179.304,8.991,149.558
C07921=1114.327,169.020,-63.515,-179.302,8.994,149.558
C07922=1114.322,169.269,-63.538,-179.299,8.998,149.558
C07923=1114.318,169.518,-63.562,-179.298,9.000,149.558
C07924=1114.314,169.767,-63.584,-179.295,9.003,149.558
C07925=1114.309,170.016,-63.608,-179.292,9.006,149.558
C07926=1114.304,170.265,-63.631,-179.291,9.009,149.558
C07927=1114.300,170.514,-63.655,-179.289,9.012,149.559
C07928=1114.295,170.763,-63.678,-179.286,9.015,149.559
C07929=1114.291,171.012,-63.701,-179.283,9.019,149.559
C07930=1114.286,171.261,-63.724,-179.282,9.021,149.559
C07931=1114.282,171.509,-63.748,-179.279,9.024,149.559
C07932=1114.277,171.758,-63.771,-179.277,9.027,149.559
C07933=1114.272,172.007,-63.795,-179.275,9.030,149.559
C07934=1114.267,172.256,-63.818,-179.273,9.033,149.559
C07935=1114.262,172.505,-63.841,-179.270,9.036,149.559
C07936=1114.259,172.718,-63.861,-179.269,9.039,149.560
C07937=1114.255,172.931,-63.881,-179.267,9.041,149.560
C07938=1114.252,173.145,-63.902,-179.265,9.044,149.560
C07939=1114.247,173.359,-63.922,-179.263,9.046,149.560
C07940=1114.244,173.573,-63.942,-179.261,9.050,149.560
C07941=1114.240,173.786,-63.962,-179.259,9.052,149.560
C07942=1114.236,174.000,-63.983,-179.257,9.054,149.560
C07943=1114.232,174.213,-64.003,-179.256,9.057,149.560
C07944=1114.227,174.462,-64.026,-179.253,9.060,149.560
C07945=1114.223,174.711,-64.050,-179.252,9.062,149.560
C07946=1114.218,174.960,-64.073,-179.249,9.065,149.560
C07947=1114.213,175.209,-64.097,-179.247,9.069,149.561
C07948=1114.209,175.458,-64.120,-179.245,9.071,149.561
C07949=1114.204,175.706,-64.144,-179.243,9.074,149.561
C07950=1114.200,175.955,-64.167,-179.240,9.078,149.561
C07951=1114.195,176.204,-64.191,-179.239,9.080,149.561
C07952=1114.191,176.453,-64.215,-179.236,9.083,149.561
C07953=1114.187,176.701,-64.238,-179.234,9.087,149.561
C07954=1114.181,176.950,-64.262,-179.232,9.089,149.561
C07955=1114.177,177.199,-64.286,-179.230,9.092,149.561
C07956=1114.172,177.448,-64.309,-179.227,9.096,149.562
C07957=1114.168,177.697,-64.333,-179.226,9.098,149.562
C07958=1114.163,177.946,-64.356,-179.223,9.101,149.562
C07959=1114.159,178.194,-64.381,-179.221,9.105,149.562
C07960=1114.154,178.444,-64.404,-179.219,9.107,149.562
C07961=1114.150,178.692,-64.428,-179.217,9.110,149.562
C07962=1114.145,178.941,-64.452,-179.215,9.113,149.562
C07963=1114.141,179.190,-64.476,-179.213,9.116,149.562
C07964=1114.136,179.439,-64.499,-179.210,9.119,149.562
C07965=1114.132,179.687,-64.523,-179.207,9.122,149.562
C07966=1114.127,179.936,-64.547,-179.205,9.125,149.562
C07967=1114.123,180.184,-64.571,-179.202,9.128,149.562
C07968=1114.119,180.434,-64.594,-179.200,9.131,149.562
C07969=1114.114,180.683,-64.618,-179.197,9.135,149.563
C07970=1114.109,180.931,-64.643,-179.195,9.138,149.563
C07971=1114.104,181.180,-64.667,-179.192,9.141,149.563
C07972=1114.100,181.429,-64.691,-179.190,9.144,149.563
C07973=1114.095,181.678,-64.714,-179.187,9.147,149.563
C07974=1114.092,181.927,-64.738,-179.185,9.150,149.563
C07975=1114.087,182.175,-64.762,-179.182,9.153,149.563
C07976=1114.082,182.425,-64.786,-179.180,9.156,149.563
C07977=1114.077,182.673,-64.810,-179.178,9.159,149.563
C07978=1114.073,182.921,-64.835,-179.175,9.162,149.563
C07979=1114.068,183.171,-64.858,-179.173,9.165,149.563
C07980=1114.064,183.420,-64.882,-179.170,9.168,149.563
C07981=1114.059,183.668,-64.907,-179.168,9.171,149.563
C07982=1114.055,183.917,-64.931,-179.165,9.174,149.563
C07983=1114.050,184.166,-64.954,-179.163,9.177,149.563
C07984=1114.046,184.414,-64.979,-179.161,9.180,149.563
C07985=1114.041,184.664,-65.004,-179.158,9.183,149.563
C07986=1114.037,184.912,-65.028,-179.156,9.186,149.563
C07987=1114.032,185.160,-65.052,-179.154,9.188,149.563
C07988=1114.028,185.409,-65.075,-179.151,9.191,149.563
C07989=1114.023,185.659,-65.100,-179.149,9.194,149.563
C07990=1114.019,185.907,-65.124,-179.146,9.198,149.563
C07991=1114.014,186.156,-65.148,-179.144,9.200,149.563
C07992=1114.010,186.369,-65.169,-179.142,9.203,149.564
C07993=1114.006,186.584,-65.190,-179.140,9.205,149.563
C07994=1114.003,186.796,-65.211,-179.138,9.207,149.563
C07995=1113.999,187.010,-65.232,-179.136,9.210,149.563
C07996=1113.994,187.223,-65.253,-179.134,9.212,149.563
C07997=1113.992,187.437,-65.274,-179.132,9.214,149.563
C07998=1113.987,187.651,-65.294,-179.130,9.217,149.564
C07999=1113.983,187.864,-65.315,-179.128,9.220,149.564
C08000=1113.978,188.112,-65.339,-179.126,9.222,149.564
C08001=1113.975,188.361,-65.364,-179.123,9.225,149.564
C08002=1113.970,188.610,-65.388,-179.121,9.227,149.564
C08003=1113.965,188.858,-65.413,-179.119,9.231,149.564
C08004=1113.960,189.107,-65.437,-179.116,9.234,149.564
C08005=1113.956,189.356,-65.462,-179.114,9.236,149.564
C08006=1113.951,189.605,-65.486,-179.112,9.239,149.564
C08007=1113.947,189.853,-65.510,-179.110,9.241,149.564
C08008=1113.943,190.103,-65.535,-179.107,9.245,149.564
C08009=1113.938,190.351,-65.559,-179.105,9.247,149.564
C08010=1113.933,190.600,-65.584,-179.103,9.250,149.564
C08011=1113.929,190.849,-65.609,-179.100,9.253,149.564
C08012=1113.924,191.097,-65.633,-179.099,9.255,149.564
C08013=1113.920,191.346,-65.658,-179.096,9.259,149.564
C08014=1113.916,191.595,-65.682,-179.095,9.261,149.564
C08015=1113.911,191.843,-65.707,-179.092,9.264,149.564
C08016=1113.907,192.093,-65.732,-179.090,9.267,149.565
C08017=1113.902,192.341,-65.756,-179.088,9.270,149.565
C08018=1113.897,192.590,-65.780,-179.086,9.272,149.565
C08019=1113.893,192.839,-65.805,-179.083,9.275,149.565
C08020=1113.889,193.087,-65.830,-179.081,9.278,149.565
C08021=1113.884,193.336,-65.855,-179.079,9.281,149.565
C08022=1113.880,193.585,-65.879,-179.077,9.283,149.565
C08023=1113.875,193.833,-65.904,-179.075,9.286,149.565
C08024=1113.870,194.083,-65.929,-179.073,9.289,149.565
C08025=1113.866,194.331,-65.954,-179.071,9.292,149.565
C08026=1113.861,194.579,-65.978,-179.069,9.295,149.565
C08027=1113.857,194.828,-66.003,-179.067,9.297,149.565
C08028=1113.852,195.077,-66.028,-179.065,9.300,149.565
C08029=1113.849,195.326,-66.053,-179.063,9.303,149.566
C08030=1113.843,195.574,-66.077,-179.061,9.305,149.566
C08031=1113.839,195.824,-66.102,-179.059,9.309,149.566
C08032=1113.835,196.072,-66.127,-179.057,9.311,149.566
C08033=1113.830,196.321,-66.152,-179.055,9.314,149.566
C08034=1113.826,196.569,-66.176,-179.052,9.317,149.566
C08035=1113.821,196.818,-66.202,-179.050,9.320,149.566
C08036=1113.817,197.067,-66.227,-179.047,9.323,149.566
C08037=1113.812,197.315,-66.251,-179.044,9.327,149.566
C08038=1113.808,197.564,-66.277,-179.041,9.330,149.566
C08039=1113.803,197.813,-66.301,-179.038,9.333,149.566
C08040=1113.799,198.062,-66.326,-179.036,9.336,149.566
C08041=1113.794,198.310,-66.351,-179.033,9.339,149.566
C08042=1113.790,198.560,-66.376,-179.030,9.343,149.566
C08043=1113.785,198.808,-66.401,-179.027,9.346,149.566
C08044=1113.781,199.057,-66.426,-179.024,9.349,149.566
C08045=1113.776,199.305,-66.451,-179.021,9.351,149.566
C08046=1113.772,199.554,-66.476,-179.019,9.355,149.566
C08047=1113.768,199.802,-66.501,-179.015,9.358,149.566
C08048=1113.764,200.016,-66.523,-179.013,9.360,149.566
C08049=1113.760,200.229,-66.544,-179.010,9.363,149.566
C08050=1113.756,200.443,-66.566,-179.009,9.365,149.566
C08051=1113.752,200.656,-66.587,-179.006,9.368,149.566
C08052=1113.749,200.869,-66.609,-179.004,9.371,149.566
C08053=1113.745,201.082,-66.630,-179.001,9.373,149.566
C08054=1113.741,201.296,-66.653,-178.999,9.376,149.566
C08055=1113.736,201.509,-66.674,-178.996,9.378,149.565
C08056=1113.733,201.758,-66.699,-178.993,9.381,149.565
C08057=1113.728,202.007,-66.724,-178.990,9.384,149.565
C08058=1113.724,202.255,-66.750,-178.987,9.387,149.565
C08059=1113.719,202.504,-66.775,-178.985,9.390,149.565
C08060=1113.714,202.753,-66.800,-178.982,9.393,149.565
C08061=1113.711,203.001,-66.825,-178.979,9.396,149.565
C08062=1113.706,203.250,-66.851,-178.975,9.399,149.565
C08063=1113.701,203.499,-66.876,-178.973,9.402,149.565
C08064=1113.697,203.747,-66.901,-178.970,9.405,149.565
C08065=1113.692,203.996,-66.927,-178.967,9.408,149.565
C08066=1113.688,204.245,-66.953,-178.964,9.411,149.565
C08067=1113.683,204.493,-66.977,-178.962,9.414,149.564
C08068=1113.679,204.742,-67.003,-178.959,9.416,149.564
C08069=1113.675,204.991,-67.029,-178.956,9.419,149.564
C08070=1113.670,205.239,-67.054,-178.953,9.422,149.564
C08071=1113.666,205.488,-67.080,-178.950,9.425,149.564
C08072=1113.661,205.737,-67.105,-178.947,9.428,149.564
C08073=1113.656,205.985,-67.130,-178.944,9.430,149.564
C08074=1113.652,206.234,-67.156,-178.942,9.433,149.564
C08075=1113.648,206.483,-67.182,-178.939,9.436,149.564
C08076=1113.643,206.731,-67.207,-178.936,9.439,149.564
C08077=1113.639,206.980,-67.233,-178.933,9.442,149.563
C08078=1113.634,207.229,-67.259,-178.930,9.445,149.564
C08079=1113.630,207.477,-67.284,-178.927,9.448,149.563
C08080=1113.625,207.726,-67.310,-178.924,9.451,149.563
C08081=1113.621,207.974,-67.336,-178.921,9.454,149.563
C08082=1113.617,208.223,-67.361,-178.918,9.457,149.563
C08083=1113.612,208.471,-67.387,-178.915,9.460,149.563
C08084=1113.608,208.720,-67.413,-178.913,9.463,149.563
C08085=1113.604,208.969,-67.438,-178.910,9.465,149.563
C08086=1113.599,209.217,-67.464,-178.907,9.468,149.563
C08087=1113.595,209.466,-67.489,-178.904,9.471,149.563
C08088=1113.590,209.715,-67.515,-178.902,9.474,149.563
C08089=1113.585,209.964,-67.542,-178.899,9.477,149.563
C08090=1113.581,210.212,-67.567,-178.896,9.480,149.563
C08091=1113.576,210.461,-67.593,-178.894,9.483,149.563
C08092=1113.572,210.710,-67.618,-178.890,9.487,149.563
C08093=1113.568,210.958,-67.644,-178.887,9.490,149.563
C08094=1113.564,211.207,-67.670,-178.884,9.492,149.563
C08095=1113.558,211.455,-67.697,-178.882,9.496,149.563
C08096=1113.554,211.704,-67.722,-178.879,9.498,149.562
C08097=1113.550,211.953,-67.748,-178.876,9.501,149.562
C08098=1113.546,212.201,-67.774,-178.874,9.505,149.563
C08099=1113.542,212.450,-67.800,-178.871,9.507,149.562
C08100=1113.537,212.698,-67.826,-178.868,9.511,149.562
C08101=1113.532,212.947,-67.852,-178.865,9.514,149.563
C08102=1113.528,213.196,-67.878,-178.863,9.517,149.563
C08103=1113.524,213.444,-67.904,-178.860,9.520,149.563
C08104=1113.520,213.658,-67.926,-178.858,9.523,149.563
C08105=1113.516,213.871,-67.948,-178.856,9.525,149.563
C08106=1113.513,214.083,-67.971,-178.855,9.527,149.563
C08107=1113.509,214.297,-67.994,-178.853,9.530,149.563
C08108=1113.505,214.510,-68.016,-178.851,9.533,149.563
C08109=1113.501,214.723,-68.039,-178.849,9.536,149.563
C08110=1113.497,214.937,-68.061,-178.847,9.538,149.563
C08111=1113.494,215.149,-68.083,-178.845,9.540,149.563
C08112=1113.489,215.398,-68.109,-178.843,9.543,149.564
C08113=1113.485,215.647,-68.135,-178.841,9.546,149.564
C08114=1113.480,215.895,-68.161,-178.838,9.549,149.564
C08115=1113.475,216.144,-68.187,-178.837,9.552,149.564
C08116=1113.472,216.393,-68.214,-178.834,9.555,149.564
C08117=1113.467,216.641,-68.240,-178.832,9.558,149.564
C08118=1113.463,216.890,-68.267,-178.829,9.561,149.564
C08119=1113.458,217.139,-68.293,-178.827,9.564,149.564
C08120=1113.454,217.387,-68.319,-178.825,9.567,149.564
C08121=1113.450,217.636,-68.345,-178.823,9.570,149.564
C08122=1113.445,217.884,-68.371,-178.820,9.573,149.565
C08123=1113.440,218.133,-68.398,-178.818,9.576,149.565
C08124=1113.436,218.381,-68.424,-178.816,9.579,149.565
C08125=1113.432,218.630,-68.450,-178.814,9.582,149.565
C08126=1113.427,218.878,-68.477,-178.811,9.585,149.565
C08127=1113.423,219.127,-68.503,-178.809,9.588,149.565
C08128=1113.418,219.375,-68.530,-178.807,9.591,149.565
C08129=1113.414,219.624,-68.556,-178.805,9.594,149.565
C08130=1113.410,219.872,-68.582,-178.802,9.597,149.565
C08131=1113.406,220.121,-68.609,-178.800,9.600,149.565
C08132=1113.401,220.370,-68.635,-178.797,9.604,149.566
C08133=1113.397,220.618,-68.662,-178.795,9.607,149.566
C08134=1113.392,220.867,-68.688,-178.792,9.610,149.566
C08135=1113.388,221.115,-68.715,-178.790,9.613,149.566
C08136=1113.384,221.364,-68.741,-178.787,9.616,149.566
C08137=1113.379,221.613,-68.768,-178.785,9.619,149.566
C08138=1113.375,221.861,-68.794,-178.783,9.622,149.566
C08139=1113.370,222.109,-68.821,-178.781,9.625,149.566
C08140=1113.366,222.358,-68.847,-178.778,9.628,149.566
C08141=1113.361,222.607,-68.874,-178.775,9.631,149.566
C08142=1113.358,222.855,-68.900,-178.773,9.634,149.566
C08143=1113.353,223.103,-68.927,-178.770,9.637,149.566
C08144=1113.348,223.353,-68.954,-178.768,9.640,149.567
C08145=1113.344,223.601,-68.980,-178.765,9.644,149.567
C08146=1113.339,223.849,-69.007,-178.763,9.647,149.567
C08147=1113.335,224.097,-69.034,-178.760,9.650,149.567
C08148=1113.331,224.346,-69.061,-178.758,9.653,149.567
C08149=1113.326,224.595,-69.087,-178.755,9.656,149.567
C08150=1113.322,224.844,-69.114,-178.753,9.659,149.567
C08151=1113.318,225.092,-69.141,-178.750,9.662,149.567
C08152=1113.314,225.341,-69.168,-178.747,9.665,149.567
C08153=1113.309,225.589,-69.195,-178.744,9.669,149.567
C08154=1113.305,225.838,-69.222,-178.742,9.672,149.567
C08155=1113.301,226.086,-69.248,-178.739,9.675,149.567
C08156=1113.296,226.334,-69.275,-178.736,9.678,149.567
C08157=1113.291,226.583,-69.302,-178.734,9.681,149.567
C08158=1113.287,226.832,-69.328,-178.731,9.684,149.567
C08159=1113.282,227.080,-69.355,-178.729,9.687,149.567
C08160=1113.279,227.293,-69.379,-178.726,9.689,149.567
C08161=1113.275,227.506,-69.402,-178.724,9.692,149.567
C08162=1113.272,227.719,-69.424,-178.721,9.695,149.567
C08163=1113.268,227.932,-69.448,-178.719,9.697,149.567
C08164=1113.264,228.145,-69.471,-178.716,9.700,149.567
C08165=1113.260,228.359,-69.494,-178.714,9.702,149.567
C08166=1113.256,228.572,-69.518,-178.712,9.705,149.567
C08167=1113.253,228.785,-69.540,-178.710,9.708,149.567
C08168=1113.249,229.033,-69.568,-178.707,9.711,149.567
C08169=1113.244,229.282,-69.595,-178.704,9.714,149.567
C08170=1113.240,229.530,-69.622,-178.701,9.717,149.567
C08171=1113.235,229.779,-69.649,-178.698,9.720,149.567
C08172=1113.232,230.028,-69.676,-178.695,9.723,149.567
C08173=1113.227,230.276,-69.703,-178.692,9.726,149.567
C08174=1113.223,230.524,-69.730,-178.689,9.729,149.567
C08175=1113.218,230.773,-69.757,-178.687,9.732,149.567
C08176=1113.213,231.021,-69.785,-178.684,9.734,149.567
C08177=1113.210,231.270,-69.811,-178.681,9.737,149.566
C08178=1113.205,231.518,-69.838,-178.678,9.740,149.567
C08179=1113.201,231.766,-69.866,-178.675,9.743,149.566
C08180=1113.196,232.015,-69.893,-178.672,9.746,149.566
C08181=1113.192,232.263,-69.920,-178.669,9.749,149.566
C08182=1113.188,232.513,-69.948,-178.667,9.752,149.566
C08183=1113.183,232.760,-69.976,-178.664,9.754,149.566
C08184=1113.179,233.009,-70.003,-178.661,9.757,149.566
C08185=1113.174,233.257,-70.030,-178.658,9.760,149.566
C08186=1113.171,233.506,-70.057,-178.655,9.763,149.566
C08187=1113.166,233.754,-70.084,-178.653,9.766,149.566
C08188=1113.162,234.003,-70.111,-178.650,9.768,149.566
C08189=1113.158,234.251,-70.139,-178.647,9.771,149.566
C08190=1113.153,234.500,-70.167,-178.644,9.773,149.565
C08191=1113.148,234.748,-70.194,-178.641,9.776,149.565
C08192=1113.144,234.996,-70.221,-178.639,9.779,149.565
C08193=1113.140,235.245,-70.249,-178.636,9.782,149.565
C08194=1113.136,235.493,-70.277,-178.633,9.785,149.565
C08195=1113.131,235.742,-70.304,-178.631,9.787,149.565
C08196=1113.127,235.990,-70.332,-178.628,9.789,149.565
C08197=1113.123,236.239,-70.359,-178.625,9.792,149.565
C08198=1113.118,236.487,-70.386,-178.622,9.795,149.565
C08199=1113.114,236.736,-70.414,-178.620,9.797,149.565
C08200=1113.110,236.984,-70.441,-178.617,9.800,149.565
C08201=1113.105,237.232,-70.469,-178.614,9.803,149.564
C08202=1113.101,237.481,-70.496,-178.611,9.805,149.564
C08203=1113.097,237.729,-70.524,-178.609,9.808,149.564
C08204=1113.092,237.977,-70.552,-178.606,9.810,149.564
C08205=1113.088,238.227,-70.580,-178.603,9.813,149.564
C08206=1113.083,238.475,-70.608,-178.601,9.815,149.564
C08207=1113.079,238.724,-70.635,-178.599,9.818,149.564
C08208=1113.075,238.972,-70.663,-178.596,9.821,149.564
C08209=1113.071,239.219,-70.691,-178.593,9.823,149.564
C08210=1113.067,239.469,-70.718,-178.590,9.826,149.564
C08211=1113.062,239.717,-70.746,-178.588,9.828,149.564
C08212=1113.058,239.966,-70.773,-178.585,9.831,149.564
C08213=1113.053,240.214,-70.802,-178.583,9.834,149.563
C08214=1113.049,240.462,-70.829,-178.581,9.836,149.564
C08215=1113.045,240.711,-70.857,-178.578,9.839,149.563
C08216=1113.041,240.923,-70.881,-178.575,9.841,149.563
C08217=1113.037,241.136,-70.905,-178.573,9.843,149.563
C08218=1113.034,241.349,-70.928,-178.571,9.845,149.563
C08219=1113.030,241.562,-70.953,-178.569,9.847,149.563
C08220=1113.026,241.775,-70.976,-178.567,9.849,149.563
C08221=1113.022,241.988,-71.000,-178.565,9.852,149.563
C08222=1113.019,242.201,-71.024,-178.563,9.854,149.563
C08223=1113.016,242.414,-71.048,-178.561,9.856,149.563
C08224=1113.011,242.662,-71.076,-178.558,9.859,149.563
C08225=1113.007,242.911,-71.104,-178.556,9.861,149.563
C08226=1113.002,243.160,-71.132,-178.553,9.864,149.563
C08227=1112.998,243.408,-71.160,-178.551,9.866,149.563
C08228=1112.994,243.656,-71.187,-178.549,9.869,149.563
C08229=1112.989,243.904,-71.216,-178.546,9.871,149.563
C08230=1112.985,244.153,-71.244,-178.544,9.874,149.563
C08231=1112.981,244.401,-71.272,-178.541,9.876,149.563
C08232=1112.976,244.650,-71.301,-178.539,9.879,149.563
C08233=1112.972,244.898,-71.328,-178.537,9.882,149.563
C08234=1112.968,245.147,-71.356,-178.535,9.885,149.563
C08235=1112.964,245.394,-71.383,-178.532,9.887,149.563
C08236=1112.959,245.643,-71.412,-178.530,9.889,149.563
C08237=1112.955,245.891,-71.440,-178.528,9.892,149.563
C08238=1112.951,246.140,-71.468,-178.526,9.895,149.563
C08239=1112.946,246.388,-71.497,-178.523,9.898,149.563
C08240=1112.942,246.637,-71.525,-178.522,9.900,149.563
C08241=1112.938,246.885,-71.553,-178.519,9.903,149.563
C08242=1112.933,247.133,-71.581,-178.517,9.905,149.563
C08243=1112.930,247.382,-71.609,-178.514,9.908,149.563
C08244=1112.924,247.630,-71.638,-178.512,9.911,149.563
C08245=1112.921,247.879,-71.666,-178.508,9.915,149.563
C08246=1112.916,248.127,-71.694,-178.504,9.918,149.563
C08247=1112.912,248.375,-71.722,-178.500,9.922,149.563
C08248=1112.907,248.623,-71.750,-178.497,9.925,149.563
C08249=1112.903,248.872,-71.779,-178.493,9.928,149.563
C08250=1112.899,249.121,-71.807,-178.489,9.932,149.562
C08251=1112.894,249.368,-71.836,-178.485,9.935,149.562
C08252=1112.891,249.617,-71.864,-178.482,9.938,149.562
C08253=1112.886,249.865,-71.892,-178.478,9.941,149.562
C08254=1112.882,250.114,-71.921,-178.475,9.944,149.562
C08255=1112.878,250.362,-71.949,-178.471,9.947,149.561
C08256=1112.873,250.610,-71.978,-178.469,9.950,149.561
C08257=1112.870,250.858,-72.006,-178.466,9.952,149.561
C08258=1112.865,251.107,-72.035,-178.462,9.955,149.561
C08259=1112.861,251.355,-72.063,-178.459,9.957,149.561
C08260=1112.857,251.603,-72.092,-178.456,9.960,149.560
C08261=1112.852,251.852,-72.121,-178.453,9.963,149.560
C08262=1112.848,252.100,-72.149,-178.450,9.965,149.560
C08263=1112.843,252.349,-72.177,-178.448,9.967,149.560
C08264=1112.840,252.597,-72.206,-178.444,9.970,149.560
C08265=1112.835,252.845,-72.235,-178.442,9.972,149.560
C08266=1112.831,253.094,-72.263,-178.439,9.975,149.559
C08267=1112.827,253.342,-72.292,-178.437,9.976,149.559
C08268=1112.822,253.590,-72.321,-178.434,9.979,149.559
C08269=1112.818,253.838,-72.349,-178.432,9.981,149.559
C08270=1112.814,254.087,-72.378,-178.429,9.983,149.559
C08271=1112.809,254.335,-72.406,-178.427,9.986,149.559
C08272=1112.806,254.548,-72.431,-178.425,9.988,149.559
C08273=1112.802,254.761,-72.456,-178.423,9.990,149.559
C08274=1112.798,254.974,-72.480,-178.421,9.991,149.559
C08275=1112.795,255.187,-72.505,-178.420,9.993,149.559
C08276=1112.791,255.399,-72.530,-178.418,9.995,149.559
C08277=1112.787,255.612,-72.554,-178.416,9.997,149.559
C08278=1112.784,255.825,-72.579,-178.415,9.998,149.559
C08279=1112.780,256.038,-72.604,-178.413,10.000,149.559
C08280=1112.776,256.286,-72.633,-178.411,10.003,149.559
C08281=1112.772,256.534,-72.661,-178.408,10.006,149.559
C08282=1112.767,256.782,-72.690,-178.405,10.009,149.559
C08283=1112.763,257.031,-72.719,-178.403,10.012,149.559
C08284=1112.759,257.279,-72.748,-178.400,10.015,149.559
C08285=1112.754,257.527,-72.776,-178.397,10.017,149.559
C08286=1112.750,257.776,-72.806,-178.394,10.020,149.558
C08287=1112.746,258.024,-72.835,-178.391,10.023,149.558
C08288=1112.742,258.272,-72.863,-178.388,10.026,149.558
C08289=1112.737,258.520,-72.893,-178.385,10.029,149.558
C08290=1112.733,258.769,-72.921,-178.382,10.031,149.558
C08291=1112.729,259.017,-72.951,-178.380,10.033,149.558
C08292=1112.725,259.265,-72.980,-178.377,10.036,149.558
C08293=1112.721,259.514,-73.008,-178.374,10.039,149.558
C08294=1112.717,259.762,-73.038,-178.372,10.042,149.558
C08295=1112.712,260.010,-73.067,-178.369,10.045,149.558
C08296=1112.707,260.259,-73.096,-178.366,10.048,149.558
C08297=1112.704,260.507,-73.124,-178.363,10.050,149.558
C08298=1112.700,260.755,-73.154,-178.360,10.053,149.558
C08299=1112.695,261.004,-73.183,-178.357,10.056,149.557
C08300=1112.691,261.251,-73.212,-178.354,10.059,149.557
C08301=1112.686,261.500,-73.241,-178.351,10.061,149.557
C08302=1112.682,261.748,-73.271,-178.348,10.064,149.557
C08303=1112.678,261.996,-73.300,-178.345,10.067,149.557
C08304=1112.674,262.245,-73.328,-178.342,10.070,149.557
C08305=1112.670,262.493,-73.358,-178.339,10.072,149.557
C08306=1112.666,262.741,-73.387,-178.336,10.075,149.557
C08307=1112.662,262.990,-73.417,-178.332,10.078,149.556
C08308=1112.657,263.237,-73.446,-178.329,10.081,149.556
C08309=1112.653,263.485,-73.475,-178.327,10.084,149.556
C08310=1112.649,263.734,-73.505,-178.324,10.087,149.556
C08311=1112.644,263.983,-73.533,-178.320,10.089,149.556
C08312=1112.640,264.231,-73.563,-178.317,10.092,149.556
C08313=1112.636,264.479,-73.592,-178.314,10.094,149.556
C08314=1112.632,264.727,-73.622,-178.311,10.097,149.555
C08315=1112.627,264.976,-73.651,-178.309,10.099,149.555
C08316=1112.623,265.224,-73.681,-178.306,10.102,149.555
C08317=1112.619,265.472,-73.710,-178.303,10.104,149.555
C08318=1112.614,265.720,-73.739,-178.301,10.106,149.555
C08319=1112.610,265.968,-73.769,-178.298,10.109,149.555
C08320=1112.606,266.216,-73.798,-178.295,10.112,149.555
C08321=1112.602,266.465,-73.828,-178.292,10.114,149.555
C08322=1112.597,266.713,-73.857,-178.289,10.117,149.554
C08323=1112.593,266.961,-73.886,-178.286,10.119,149.554
C08324=1112.589,267.209,-73.917,-178.284,10.121,149.554
C08325=1112.585,267.457,-73.946,-178.281,10.124,149.554
C08326=1112.581,267.705,-73.975,-178.278,10.127,149.554
C08327=1112.576,267.954,-74.006,-178.275,10.130,149.554
C08328=1112.573,268.167,-74.030,-178.273,10.132,149.554
C08329=1112.569,268.379,-74.056,-178.271,10.134,149.554
C08330=1112.566,268.592,-74.082,-178.268,10.136,149.554
C08331=1112.562,268.804,-74.106,-178.265,10.138,149.553
C08332=1112.559,269.017,-74.132,-178.264,10.141,149.554
C08333=1112.555,269.229,-74.158,-178.261,10.143,149.553
C08334=1112.551,269.443,-74.183,-178.259,10.145,149.553
C08335=1112.547,269.655,-74.209,-178.256,10.147,149.553
C08336=1112.543,269.903,-74.238,-178.254,10.149,149.553
C08337=1112.539,270.151,-74.267,-178.251,10.152,149.553
C08338=1112.535,270.399,-74.298,-178.248,10.155,149.553
C08339=1112.531,270.648,-74.328,-178.245,10.158,149.553
C08340=1112.527,270.897,-74.357,-178.242,10.160,149.553
C08341=1112.523,271.145,-74.387,-178.240,10.162,149.553
C08342=1112.519,271.393,-74.417,-178.237,10.165,149.552
C08343=1112.515,271.641,-74.447,-178.234,10.168,149.552
C08344=1112.510,271.889,-74.477,-178.231,10.171,149.552
C08345=1112.506,272.137,-74.507,-178.228,10.173,149.552
C08346=1112.502,272.385,-74.536,-178.225,10.176,149.552
C08347=1112.497,272.634,-74.566,-178.222,10.178,149.552
C08348=1112.493,272.881,-74.596,-178.219,10.181,149.552
C08349=1112.489,273.130,-74.626,-178.216,10.183,149.552
C08350=1112.485,273.377,-74.656,-178.213,10.186,149.551
C08351=1112.481,273.626,-74.685,-178.211,10.189,149.551
C08352=1112.476,273.874,-74.717,-178.208,10.192,149.551
C08353=1112.472,274.123,-74.746,-178.205,10.194,149.551
C08354=1112.468,274.371,-74.776,-178.202,10.197,149.551
C08355=1112.464,274.619,-74.806,-178.199,10.199,149.551
C08356=1112.459,274.867,-74.836,-178.196,10.202,149.551
C08357=1112.455,275.115,-74.866,-178.193,10.204,149.551
C08358=1112.451,275.363,-74.896,-178.190,10.207,149.550
C08359=1112.447,275.612,-74.926,-178.187,10.210,149.550
C08360=1112.443,275.859,-74.957,-178.184,10.213,149.550
C08361=1112.438,276.108,-74.987,-178.181,10.215,149.550
C08362=1112.435,276.356,-75.017,-178.178,10.218,149.550
C08363=1112.430,276.604,-75.046,-178.175,10.221,149.550
C08364=1112.426,276.852,-75.077,-178.172,10.223,149.550
C08365=1112.423,277.100,-75.108,-178.169,10.226,149.550
C08366=1112.418,277.349,-75.138,-178.167,10.228,149.549
C08367=1112.414,277.596,-75.168,-178.164,10.231,149.549
C08368=1112.410,277.844,-75.198,-178.161,10.233,149.549
C08369=1112.405,278.093,-75.228,-178.158,10.236,149.549
C08370=1112.402,278.341,-75.259,-178.155,10.239,149.549
C08371=1112.397,278.589,-75.289,-178.151,10.241,149.549
C08372=1112.393,278.837,-75.319,-178.149,10.244,149.549
C08373=1112.388,279.085,-75.350,-178.146,10.247,149.548
C08374=1112.385,279.333,-75.380,-178.142,10.249,149.548
C08375=1112.380,279.581,-75.411,-178.139,10.252,149.548
C08376=1112.376,279.830,-75.440,-178.136,10.255,149.548
C08377=1112.372,280.078,-75.471,-178.133,10.257,149.548
C08378=1112.368,280.326,-75.502,-178.130,10.260,149.548
C08379=1112.364,280.574,-75.532,-178.127,10.263,149.547
C08380=1112.360,280.822,-75.563,-178.124,10.265,149.547
C08381=1112.355,281.070,-75.593,-178.121,10.268,149.547
C08382=1112.352,281.319,-75.623,-178.118,10.270,149.547
C08383=1112.347,281.566,-75.654,-178.115,10.273,149.547
C08384=1112.344,281.779,-75.680,-178.112,10.275,149.547
C08385=1112.339,281.991,-75.707,-178.110,10.277,149.546
C08386=1112.336,282.204,-75.733,-178.107,10.279,149.546
C08387=1112.333,282.417,-75.758,-178.104,10.281,149.546
C08388=1112.329,282.630,-75.785,-178.102,10.283,149.546
C08389=1112.325,282.841,-75.811,-178.099,10.286,149.546
C08390=1112.322,283.054,-75.837,-178.096,10.288,149.546
C08391=1112.318,283.267,-75.864,-178.094,10.290,149.545
C08392=1112.314,283.515,-75.894,-178.091,10.293,149.545
C08393=1112.310,283.763,-75.924,-178.088,10.295,149.545
C08394=1112.306,284.011,-75.956,-178.085,10.298,149.545
C08395=1112.302,284.259,-75.986,-178.082,10.300,149.545
C08396=1112.297,284.507,-76.017,-178.079,10.303,149.545
C08397=1112.293,284.756,-76.048,-178.076,10.306,149.545
C08398=1112.290,285.003,-76.079,-178.073,10.307,149.544
C08399=1112.285,285.251,-76.109,-178.070,10.310,149.544
C08400=1112.281,285.499,-76.140,-178.067,10.312,149.544
C08401=1112.277,285.747,-76.171,-178.064,10.315,149.544
C08402=1112.273,285.996,-76.202,-178.061,10.318,149.544
C08403=1112.268,286.244,-76.233,-178.057,10.320,149.543
C08404=1112.264,286.491,-76.263,-178.055,10.323,149.543
C08405=1112.261,286.740,-76.294,-178.051,10.326,149.543
C08406=1112.256,286.987,-76.325,-178.049,10.328,149.543
C08407=1112.252,287.236,-76.356,-178.046,10.330,149.543
C08408=1112.248,287.484,-76.387,-178.043,10.333,149.543
C08409=1112.244,287.731,-76.417,-178.040,10.336,149.542
C08410=1112.240,287.980,-76.449,-178.036,10.338,149.542
C08411=1112.235,288.227,-76.480,-178.033,10.341,149.542
C08412=1112.231,288.476,-76.511,-178.030,10.343,149.542
C08413=1112.227,288.724,-76.542,-178.027,10.346,149.542
C08414=1112.224,288.972,-76.572,-178.024,10.348,149.541
C08415=1112.219,289.220,-76.604,-178.021,10.350,149.541
C08416=1112.215,289.468,-76.635,-178.018,10.353,149.541
C08417=1112.211,289.716,-76.666,-178.015,10.356,149.541
C08418=1112.206,289.964,-76.697,-178.012,10.358,149.541
C08419=1112.202,290.212,-76.728,-178.009,10.361,149.541
C08420=1112.198,290.460,-76.759,-178.006,10.363,149.541
C08421=1112.195,290.708,-76.790,-178.003,10.366,149.540
C08422=1112.190,290.956,-76.821,-178.000,10.369,149.540
C08423=1112.186,291.204,-76.853,-177.997,10.370,149.540
C08424=1112.182,291.452,-76.884,-177.994,10.373,149.540
C08425=1112.178,291.700,-76.916,-177.991,10.375,149.540
C08426=1112.173,291.948,-76.946,-177.988,10.378,149.539
C08427=1112.169,292.197,-76.978,-177.985,10.381,149.539
C08428=1112.165,292.444,-77.009,-177.982,10.383,149.539
C08429=1112.161,292.693,-77.040,-177.979,10.386,149.539
C08430=1112.157,292.940,-77.072,-177.975,10.389,149.539
C08431=1112.153,293.189,-77.103,-177.972,10.391,149.539
C08432=1112.149,293.436,-77.134,-177.970,10.393,149.538
C08433=1112.146,293.684,-77.165,-177.967,10.396,149.538
C08434=1112.142,293.932,-77.197,-177.963,10.398,149.538
C08435=1112.137,294.180,-77.228,-177.960,10.401,149.538
C08436=1112.133,294.428,-77.259,-177.957,10.403,149.538
C08437=1112.129,294.676,-77.291,-177.954,10.406,149.538
C08438=1112.125,294.924,-77.323,-177.951,10.409,149.537
C08439=1112.121,295.172,-77.353,-177.948,10.411,149.537
C08440=1112.117,295.384,-77.381,-177.946,10.413,149.537
C08441=1112.113,295.597,-77.408,-177.943,10.415,149.537
C08442=1112.109,295.809,-77.435,-177.940,10.418,149.537
C08443=1112.107,296.021,-77.462,-177.938,10.420,149.537
C08444=1112.103,296.234,-77.489,-177.935,10.422,149.536
C08445=1112.099,296.446,-77.516,-177.932,10.424,149.536
C08446=1112.095,296.659,-77.543,-177.930,10.426,149.536
C08447=1112.093,296.871,-77.570,-177.927,10.428,149.536
C08448=1112.089,297.119,-77.602,-177.924,10.431,149.536
C08449=1112.084,297.367,-77.632,-177.921,10.433,149.536
C08450=1112.080,297.615,-77.665,-177.918,10.436,149.535
C08451=1112.076,297.863,-77.697,-177.915,10.439,149.535
C08452=1112.072,298.111,-77.728,-177.912,10.441,149.535
C08453=1112.068,298.359,-77.759,-177.909,10.444,149.535
C08454=1112.064,298.607,-77.791,-177.905,10.446,149.535
C08455=1112.060,298.855,-77.823,-177.903,10.448,149.535
C08456=1112.055,299.103,-77.855,-177.900,10.451,149.534
C08457=1112.052,299.351,-77.887,-177.897,10.453,149.534
C08458=1112.047,299.598,-77.918,-177.894,10.456,149.534
C08459=1112.044,299.846,-77.950,-177.890,10.459,149.534
C08460=1112.040,300.094,-77.982,-177.888,10.461,149.534
C08461=1112.035,300.343,-78.013,-177.884,10.464,149.534
C08462=1112.031,300.591,-78.045,-177.881,10.467,149.533
C08463=1112.027,300.839,-78.077,-177.878,10.469,149.533
C08464=1112.023,301.086,-78.109,-177.875,10.472,149.533
C08465=1112.018,301.335,-78.141,-177.872,10.473,149.533
C08466=1112.015,301.583,-78.173,-177.869,10.476,149.533
C08467=1112.010,301.830,-78.204,-177.866,10.479,149.532
C08468=1112.006,302.078,-78.237,-177.863,10.481,149.532
C08469=1112.002,302.326,-78.269,-177.860,10.484,149.532
C08470=1111.998,302.574,-78.300,-177.856,10.486,149.532
C08471=1111.993,302.822,-78.333,-177.854,10.489,149.532
C08472=1111.990,303.070,-78.364,-177.850,10.491,149.532
C08473=1111.986,303.317,-78.397,-177.847,10.494,149.531
C08474=1111.982,303.566,-78.429,-177.845,10.496,149.531
C08475=1111.978,303.813,-78.461,-177.842,10.499,149.531
C08476=1111.974,304.061,-78.493,-177.838,10.501,149.531
C08477=1111.969,304.309,-78.525,-177.835,10.504,149.531
C08478=1111.966,304.558,-78.557,-177.832,10.506,149.530
C08479=1111.961,304.805,-78.588,-177.829,10.509,149.530
C08480=1111.957,305.053,-78.622,-177.826,10.512,149.530
C08481=1111.954,305.301,-78.653,-177.823,10.514,149.530
C08482=1111.949,305.549,-78.686,-177.820,10.517,149.530
C08483=1111.945,305.796,-78.717,-177.817,10.519,149.530
C08484=1111.940,306.045,-78.750,-177.814,10.521,149.529
C08485=1111.937,306.292,-78.782,-177.811,10.524,149.529
C08486=1111.933,306.540,-78.814,-177.808,10.526,149.529
C08487=1111.929,306.788,-78.847,-177.805,10.529,149.529
C08488=1111.925,307.036,-78.879,-177.801,10.532,149.529
C08489=1111.920,307.284,-78.911,-177.798,10.534,149.529
C08490=1111.917,307.532,-78.943,-177.795,10.537,149.528
C08491=1111.913,307.779,-78.976,-177.792,10.539,149.528
C08492=1111.909,308.027,-79.008,-177.789,10.542,149.528
C08493=1111.904,308.276,-79.041,-177.786,10.544,149.528
C08494=1111.901,308.523,-79.073,-177.783,10.546,149.528
C08495=1111.896,308.771,-79.105,-177.780,10.549,149.527
C08496=1111.893,308.983,-79.134,-177.777,10.552,149.527
C08497=1111.889,309.196,-79.161,-177.775,10.554,149.527
C08498=1111.886,309.408,-79.189,-177.772,10.555,149.527
C08499=1111.882,309.620,-79.216,-177.769,10.558,149.527
C08500=1111.879,309.832,-79.244,-177.767,10.560,149.527
C08501=1111.875,310.045,-79.273,-177.764,10.562,149.527
C08502=1111.872,310.257,-79.300,-177.761,10.564,149.526
C08503=1111.868,310.469,-79.328,-177.759,10.566,149.526
C08504=1111.865,310.717,-79.360,-177.755,10.569,149.526
C08505=1111.861,310.965,-79.393,-177.753,10.572,149.526
C08506=1111.856,311.213,-79.426,-177.749,10.574,149.526
C08507=1111.853,311.461,-79.458,-177.746,10.577,149.526
C08508=1111.849,311.708,-79.491,-177.744,10.579,149.525
C08509=1111.844,311.956,-79.522,-177.740,10.581,149.525
C08510=1111.840,312.204,-79.556,-177.737,10.584,149.525
C08511=1111.836,312.451,-79.589,-177.734,10.586,149.525
C08512=1111.832,312.699,-79.621,-177.731,10.589,149.525
C08513=1111.828,312.947,-79.654,-177.728,10.591,149.525
C08514=1111.824,313.195,-79.686,-177.724,10.594,149.524
C08515=1111.820,313.443,-79.719,-177.722,10.597,149.524
C08516=1111.816,313.691,-79.752,-177.718,10.599,149.524
C08517=1111.812,313.938,-79.785,-177.715,10.602,149.524
C08518=1111.808,314.187,-79.818,-177.713,10.603,149.524
C08519=1111.804,314.434,-79.850,-177.710,10.606,149.524
C08520=1111.800,314.682,-79.883,-177.706,10.609,149.523
C08521=1111.796,314.930,-79.916,-177.703,10.611,149.523
C08522=1111.792,315.178,-79.948,-177.700,10.614,149.523
C08523=1111.788,315.425,-79.981,-177.697,10.616,149.523
C08524=1111.784,315.673,-80.015,-177.694,10.619,149.523
C08525=1111.780,315.921,-80.048,-177.690,10.622,149.522
C08526=1111.776,316.169,-80.080,-177.688,10.624,149.522
C08527=1111.772,316.416,-80.113,-177.684,10.627,149.522
C08528=1111.768,316.664,-80.146,-177.682,10.628,149.522
C08529=1111.764,316.912,-80.179,-177.679,10.631,149.522
C08530=1111.760,317.160,-80.212,-177.675,10.634,149.521
C08531=1111.757,317.408,-80.245,-177.672,10.636,149.521
C08532=1111.753,317.656,-80.278,-177.669,10.639,149.521
C08533=1111.748,317.903,-80.311,-177.666,10.641,149.521
C08534=1111.744,318.152,-80.344,-177.663,10.644,149.521
C08535=1111.740,318.399,-80.377,-177.659,10.647,149.521
C08536=1111.736,318.647,-80.410,-177.657,10.649,149.521
C08537=1111.732,318.895,-80.443,-177.653,10.652,149.520
C08538=1111.728,319.142,-80.476,-177.651,10.653,149.520
C08539=1111.724,319.390,-80.509,-177.648,10.656,149.520
C08540=1111.720,319.638,-80.542,-177.644,10.659,149.520
C08541=1111.716,319.885,-80.575,-177.641,10.661,149.519
C08542=1111.712,320.134,-80.609,-177.638,10.664,149.519
C08543=1111.708,320.381,-80.643,-177.635,10.666,149.519
C08544=1111.704,320.629,-80.676,-177.632,10.669,149.519
C08545=1111.700,320.876,-80.709,-177.628,10.672,149.519
C08546=1111.696,321.124,-80.742,-177.625,10.674,149.519
C08547=1111.692,321.372,-80.775,-177.622,10.677,149.518
C08548=1111.688,321.620,-80.809,-177.620,10.678,149.518
C08549=1111.685,321.868,-80.841,-177.616,10.681,149.518
C08550=1111.681,322.115,-80.875,-177.613,10.684,149.518
C08551=1111.677,322.363,-80.908,-177.610,10.686,149.518
C08552=1111.673,322.575,-80.937,-177.607,10.689,149.518
C08553=1111.670,322.787,-80.965,-177.604,10.691,149.517
C08554=1111.666,322.999,-80.994,-177.602,10.693,149.517
C08555=1111.663,323.211,-81.023,-177.599,10.695,149.517
C08556=1111.659,323.424,-81.051,-177.596,10.697,149.517
C08557=1111.657,323.636,-81.080,-177.594,10.699,149.517
C08558=1111.653,323.848,-81.109,-177.591,10.701,149.517
C08559=1111.649,324.060,-81.137,-177.589,10.703,149.516
C08560=1111.646,324.308,-81.170,-177.585,10.706,149.516
C08561=1111.641,324.555,-81.205,-177.582,10.709,149.516
C08562=1111.637,324.803,-81.238,-177.579,10.711,149.516
C08563=1111.633,325.051,-81.271,-177.576,10.714,149.516
C08564=1111.629,325.298,-81.305,-177.573,10.716,149.516
C08565=1111.626,325.546,-81.338,-177.570,10.718,149.515
C08566=1111.621,325.794,-81.372,-177.567,10.720,149.515
C08567=1111.618,326.041,-81.405,-177.564,10.723,149.515
C08568=1111.614,326.289,-81.439,-177.560,10.726,149.515
C08569=1111.610,326.537,-81.473,-177.557,10.728,149.515
C08570=1111.605,326.785,-81.507,-177.554,10.731,149.514
C08571=1111.601,327.033,-81.540,-177.551,10.733,149.514
C08572=1111.597,327.280,-81.574,-177.548,10.736,149.514
C08573=1111.594,327.528,-81.607,-177.545,10.739,149.514
C08574=1111.590,327.775,-81.641,-177.542,10.740,149.514
C08575=1111.585,328.023,-81.675,-177.539,10.743,149.513
C08576=1111.582,328.271,-81.709,-177.536,10.745,149.513
C08577=1111.578,328.519,-81.742,-177.532,10.748,149.513
C08578=1111.574,328.766,-81.776,-177.529,10.750,149.513
C08579=1111.570,329.014,-81.809,-177.526,10.753,149.513
C08580=1111.566,329.262,-81.844,-177.523,10.756,149.513
C08581=1111.562,329.509,-81.878,-177.519,10.758,149.512
C08582=1111.558,329.757,-81.911,-177.517,10.761,149.512
C08583=1111.554,330.005,-81.946,-177.513,10.763,149.512
C08584=1111.550,330.252,-81.979,-177.511,10.765,149.512
C08585=1111.546,330.499,-82.013,-177.508,10.768,149.512
C08586=1111.543,330.747,-82.047,-177.504,10.770,149.511
C08587=1111.538,330.995,-82.081,-177.501,10.773,149.511
C08588=1111.534,331.242,-82.115,-177.498,10.775,149.511
C08589=1111.531,331.490,-82.149,-177.495,10.778,149.511
C08590=1111.526,331.738,-82.183,-177.491,10.780,149.511
C08591=1111.522,331.985,-82.217,-177.488,10.783,149.510
C08592=1111.519,332.233,-82.251,-177.485,10.786,149.510
C08593=1111.514,332.481,-82.285,-177.482,10.788,149.510
C08594=1111.511,332.729,-82.319,-177.479,10.790,149.510
C08595=1111.507,332.976,-82.353,-177.476,10.792,149.510
C08596=1111.502,333.224,-82.387,-177.473,10.795,149.510
C08597=1111.499,333.471,-82.421,-177.470,10.797,149.509
C08598=1111.495,333.719,-82.456,-177.466,10.800,149.509
C08599=1111.491,333.967,-82.489,-177.463,10.803,149.509
C08600=1111.487,334.214,-82.523,-177.460,10.805,149.509
C08601=1111.483,334.462,-82.558,-177.457,10.808,149.509
C08602=1111.479,334.710,-82.592,-177.454,10.810,149.508
C08603=1111.475,334.957,-82.626,-177.451,10.813,149.508
C08604=1111.472,335.205,-82.661,-177.447,10.815,149.508
C08605=1111.467,335.452,-82.695,-177.445,10.817,149.508
C08606=1111.464,335.700,-82.729,-177.442,10.820,149.508
C08607=1111.460,335.947,-82.763,-177.438,10.822,149.507
C08608=1111.457,336.159,-82.793,-177.435,10.825,149.507
C08609=1111.453,336.371,-82.822,-177.433,10.827,149.507
C08610=1111.450,336.583,-82.852,-177.430,10.828,149.507
C08611=1111.446,336.796,-82.881,-177.427,10.831,149.507
C08612=1111.442,337.008,-82.910,-177.424,10.833,149.507
C08613=1111.439,337.220,-82.939,-177.422,10.835,149.506
C08614=1111.436,337.432,-82.970,-177.419,10.837,149.506
C08615=1111.432,337.643,-82.999,-177.417,10.839,149.506
C08616=1111.429,337.891,-83.033,-177.413,10.842,149.506
C08617=1111.425,338.138,-83.068,-177.410,10.844,149.506
C08618=1111.421,338.386,-83.102,-177.407,10.847,149.506
C08619=1111.417,338.634,-83.136,-177.404,10.849,149.505
C08620=1111.413,338.882,-83.171,-177.401,10.851,149.505
C08621=1111.409,339.129,-83.205,-177.398,10.853,149.505
C08622=1111.405,339.377,-83.240,-177.395,10.856,149.505
C08623=1111.401,339.624,-83.274,-177.391,10.859,149.505
C08624=1111.398,339.871,-83.309,-177.388,10.861,149.504
C08625=1111.393,340.119,-83.344,-177.385,10.864,149.504
C08626=1111.390,340.367,-83.378,-177.382,10.866,149.504
C08627=1111.385,340.614,-83.413,-177.379,10.869,149.504
C08628=1111.381,340.862,-83.447,-177.375,10.871,149.504
C08629=1111.378,341.109,-83.482,-177.372,10.874,149.503
C08630=1111.374,341.357,-83.517,-177.370,10.876,149.503
C08631=1111.370,341.605,-83.552,-177.366,10.878,149.503
C08632=1111.365,341.852,-83.586,-177.363,10.881,149.503
C08633=1111.362,342.100,-83.621,-177.360,10.883,149.503
C08634=1111.358,342.347,-83.655,-177.356,10.886,149.502
C08635=1111.354,342.595,-83.690,-177.353,10.888,149.502
C08636=1111.351,342.842,-83.725,-177.350,10.891,149.502
C08637=1111.346,343.090,-83.760,-177.347,10.893,149.502
C08638=1111.342,343.338,-83.795,-177.344,10.896,149.502
C08639=1111.338,343.585,-83.830,-177.340,10.898,149.501
C08640=1111.335,343.832,-83.864,-177.337,10.901,149.501
C08641=1111.331,344.080,-83.900,-177.335,10.903,149.501
C08642=1111.327,344.327,-83.934,-177.331,10.905,149.501
C08643=1111.323,344.575,-83.970,-177.328,10.908,149.501
C08644=1111.319,344.823,-84.004,-177.325,10.910,149.500
C08645=1111.315,345.070,-84.038,-177.322,10.913,149.500
C08646=1111.311,345.318,-84.074,-177.318,10.915,149.500
C08647=1111.307,345.565,-84.108,-177.315,10.918,149.500
C08648=1111.303,345.813,-84.144,-177.312,10.920,149.500
C08649=1111.299,346.061,-84.179,-177.308,10.923,149.499
C08650=1111.295,346.307,-84.214,-177.306,10.925,149.499
C08651=1111.292,346.555,-84.249,-177.303,10.927,149.499
C08652=1111.288,346.803,-84.284,-177.300,10.930,149.499
C08653=1111.284,347.050,-84.319,-177.296,10.932,149.499
C08654=1111.280,347.298,-84.354,-177.293,10.935,149.498
C08655=1111.276,347.545,-84.389,-177.290,10.937,149.498
C08656=1111.273,347.793,-84.425,-177.287,10.940,149.498
C08657=1111.268,348.040,-84.459,-177.283,10.942,149.498
C08658=1111.264,348.288,-84.495,-177.280,10.945,149.498
C08659=1111.261,348.535,-84.530,-177.277,10.947,149.498
C08660=1111.256,348.783,-84.565,-177.273,10.950,149.497
C08661=1111.252,349.030,-84.600,-177.271,10.951,149.497
C08662=1111.249,349.277,-84.635,-177.268,10.954,149.497
C08663=1111.246,349.525,-84.670,-177.265,10.957,149.497
C08664=1111.242,349.737,-84.701,-177.261,10.959,149.497
C08665=1111.238,349.948,-84.731,-177.259,10.961,149.496
C08666=1111.235,350.160,-84.761,-177.256,10.964,149.496
C08667=1111.231,350.372,-84.791,-177.253,10.965,149.496
C08668=1111.229,350.584,-84.822,-177.250,10.967,149.496
C08669=1111.225,350.796,-84.851,-177.247,10.970,149.496
C08670=1111.222,351.008,-84.882,-177.245,10.971,149.495
C08671=1111.219,351.220,-84.913,-177.241,10.974,149.495
C08672=1111.215,351.467,-84.948,-177.238,10.976,149.495
C08673=1111.211,351.714,-84.983,-177.235,10.979,149.495
C08674=1111.207,351.962,-85.018,-177.231,10.981,149.495
C08675=1111.203,352.210,-85.054,-177.228,10.984,149.494
C08676=1111.200,352.457,-85.089,-177.225,10.986,149.494
C08677=1111.195,352.704,-85.124,-177.222,10.989,149.494
C08678=1111.192,352.952,-85.160,-177.218,10.991,149.494
C08679=1111.188,353.199,-85.196,-177.215,10.994,149.493
C08680=1111.184,353.447,-85.231,-177.212,10.996,149.493
C08681=1111.180,353.694,-85.267,-177.208,10.998,149.493
C08682=1111.176,353.942,-85.303,-177.205,11.001,149.493
C08683=1111.173,354.189,-85.338,-177.201,11.003,149.492
C08684=1111.168,354.436,-85.373,-177.198,11.006,149.492
C08685=1111.165,354.684,-85.409,-177.195,11.008,149.492
C08686=1111.161,354.931,-85.445,-177.191,11.010,149.492
C08687=1111.157,355.179,-85.480,-177.188,11.013,149.491
C08688=1111.154,355.426,-85.516,-177.185,11.015,149.491
C08689=1111.149,355.674,-85.552,-177.181,11.018,149.491
C08690=1111.146,355.921,-85.588,-177.178,11.020,149.491
C08691=1111.142,356.168,-85.624,-177.175,11.023,149.491
C08692=1111.138,356.415,-85.659,-177.171,11.025,149.490
C08693=1111.134,356.663,-85.694,-177.168,11.027,149.490
C08694=1111.130,356.910,-85.731,-177.165,11.030,149.490
C08695=1111.126,357.158,-85.766,-177.161,11.032,149.489
C08696=1111.123,357.405,-85.802,-177.158,11.035,149.489
C08697=1111.119,357.652,-85.838,-177.155,11.037,149.489
C08698=1111.115,357.900,-85.874,-177.151,11.039,149.489
C08699=1111.111,358.148,-85.910,-177.148,11.042,149.488
C08700=1111.108,358.395,-85.946,-177.144,11.044,149.488
C08701=1111.104,358.642,-85.981,-177.141,11.047,149.488
C08702=1111.100,358.890,-86.018,-177.138,11.049,149.488
C08703=1111.096,359.137,-86.053,-177.134,11.051,149.487
C08704=1111.093,359.384,-86.089,-177.131,11.053,149.487
C08705=1111.089,359.632,-86.125,-177.128,11.056,149.487
C08706=1111.085,359.880,-86.161,-177.125,11.058,149.487
C08707=1111.081,360.126,-86.197,-177.121,11.060,149.486
C08708=1111.078,360.374,-86.233,-177.118,11.063,149.486
C08709=1111.074,360.621,-86.270,-177.114,11.065,149.486
C08710=1111.070,360.869,-86.305,-177.111,11.068,149.486
C08711=1111.066,361.116,-86.341,-177.108,11.070,149.485
C08712=1111.062,361.363,-86.378,-177.104,11.073,149.485
C08713=1111.059,361.611,-86.413,-177.101,11.075,149.485
C08714=1111.054,361.858,-86.450,-177.097,11.077,149.485
C08715=1111.051,362.106,-86.486,-177.094,11.080,149.484
C08716=1111.047,362.352,-86.522,-177.091,11.082,149.484
C08717=1111.043,362.600,-86.558,-177.088,11.085,149.484
C08718=1111.040,362.847,-86.594,-177.084,11.087,149.484
C08719=1111.035,363.095,-86.630,-177.081,11.089,149.483
C08720=1111.033,363.306,-86.661,-177.077,11.092,149.483
C08721=1111.029,363.518,-86.692,-177.075,11.093,149.483
C08722=1111.026,363.730,-86.724,-177.072,11.095,149.483
C08723=1111.023,363.941,-86.755,-177.069,11.098,149.483
C08724=1111.020,364.153,-86.786,-177.066,11.099,149.482
C08725=1111.016,364.365,-86.817,-177.063,11.102,149.482
C08726=1111.013,364.576,-86.848,-177.060,11.104,149.482
C08727=1111.010,364.788,-86.879,-177.058,11.105,149.482
C08728=1111.006,365.035,-86.915,-177.054,11.108,149.481
C08729=1111.002,365.282,-86.952,-177.051,11.110,149.481
C08730=1110.998,365.530,-86.988,-177.047,11.112,149.481
C08731=1110.995,365.778,-87.024,-177.044,11.115,149.481
C08732=1110.991,366.025,-87.061,-177.041,11.117,149.480
C08733=1110.988,366.272,-87.097,-177.037,11.120,149.480
C08734=1110.984,366.519,-87.134,-177.034,11.122,149.480
C08735=1110.980,366.767,-87.170,-177.030,11.124,149.480
C08736=1110.976,367.014,-87.207,-177.027,11.127,149.479
C08737=1110.972,367.261,-87.244,-177.024,11.129,149.479
C08738=1110.968,367.508,-87.280,-177.021,11.132,149.479
C08739=1110.965,367.756,-87.317,-177.017,11.134,149.479
C08740=1110.961,368.003,-87.353,-177.014,11.137,149.478
C08741=1110.957,368.250,-87.389,-177.010,11.139,149.478
C08742=1110.953,368.498,-87.426,-177.007,11.141,149.478
C08743=1110.950,368.744,-87.463,-177.004,11.144,149.478
C08744=1110.946,368.992,-87.499,-177.000,11.146,149.478
C08745=1110.942,369.240,-87.537,-176.997,11.149,149.477
C08746=1110.939,369.486,-87.573,-176.993,11.151,149.477
C08747=1110.935,369.734,-87.610,-176.990,11.154,149.477
C08748=1110.931,369.981,-87.647,-176.987,11.156,149.476
C08749=1110.927,370.228,-87.683,-176.983,11.159,149.476
C08750=1110.924,370.476,-87.720,-176.980,11.161,149.476
C08751=1110.920,370.723,-87.757,-176.977,11.163,149.476
C08752=1110.916,370.970,-87.794,-176.974,11.166,149.476
C08753=1110.912,371.217,-87.830,-176.970,11.168,149.475
C08754=1110.909,371.465,-87.867,-176.967,11.171,149.475
C08755=1110.905,371.712,-87.904,-176.963,11.173,149.475
C08756=1110.901,371.959,-87.941,-176.960,11.176,149.475
C08757=1110.897,372.206,-87.977,-176.957,11.178,149.474
C08758=1110.894,372.454,-88.015,-176.953,11.180,149.474
C08759=1110.890,372.701,-88.051,-176.950,11.183,149.474
C08760=1110.886,372.948,-88.088,-176.946,11.186,149.474
C08761=1110.882,373.194,-88.125,-176.943,11.189,149.474
C08762=1110.879,373.442,-88.162,-176.940,11.191,149.473
C08763=1110.875,373.690,-88.199,-176.936,11.194,149.473
C08764=1110.871,373.937,-88.236,-176.933,11.196,149.473
C08765=1110.867,374.185,-88.273,-176.929,11.198,149.473
C08766=1110.864,374.431,-88.311,-176.926,11.201,149.472
C08767=1110.860,374.678,-88.347,-176.923,11.203,149.472
C08768=1110.857,374.926,-88.384,-176.919,11.206,149.472
C08769=1110.853,375.173,-88.421,-176.916,11.208,149.472
C08770=1110.849,375.420,-88.459,-176.913,11.211,149.472
C08771=1110.845,375.668,-88.496,-176.910,11.213,149.471
C08772=1110.841,375.915,-88.533,-176.906,11.216,149.471
C08773=1110.837,376.161,-88.571,-176.903,11.218,149.471
C08774=1110.834,376.409,-88.608,-176.900,11.221,149.471
C08775=1110.830,376.657,-88.645,-176.897,11.223,149.471
C08776=1110.826,376.868,-88.676,-176.893,11.226,149.471
C08777=1110.823,377.079,-88.709,-176.891,11.228,149.470
C08778=1110.821,377.291,-88.741,-176.888,11.230,149.470
C08779=1110.817,377.502,-88.772,-176.885,11.232,149.470
C08780=1110.814,377.713,-88.804,-176.882,11.235,149.470
C08781=1110.811,377.925,-88.836,-176.880,11.237,149.470
C08782=1110.808,378.137,-88.867,-176.876,11.239,149.470
C08783=1110.804,378.349,-88.900,-176.874,11.241,149.469
C08784=1110.801,378.595,-88.938,-176.870,11.244,149.469
C08785=1110.797,378.843,-88.974,-176.867,11.247,149.469
C08786=1110.793,379.090,-89.012,-176.864,11.249,149.469
C08787=1110.789,379.337,-89.049,-176.860,11.252,149.469
C08788=1110.786,379.584,-89.087,-176.857,11.254,149.469
C08789=1110.782,379.832,-89.124,-176.854,11.257,149.469
C08790=1110.778,380.078,-89.162,-176.851,11.260,149.468
C08791=1110.775,380.325,-89.200,-176.847,11.262,149.468
C08792=1110.771,380.573,-89.236,-176.844,11.265,149.468
C08793=1110.768,380.820,-89.274,-176.840,11.268,149.468
C08794=1110.764,381.067,-89.311,-176.837,11.271,149.468
C08795=1110.760,381.314,-89.349,-176.834,11.273,149.468
C08796=1110.757,381.561,-89.387,-176.831,11.276,149.468
C08797=1110.753,381.809,-89.424,-176.828,11.278,149.467
C08798=1110.749,382.056,-89.462,-176.825,11.281,149.467
C08799=1110.745,382.303,-89.500,-176.821,11.284,149.467
C08800=1110.742,382.549,-89.538,-176.817,11.287,149.467
C08801=1110.738,382.797,-89.575,-176.815,11.290,149.467
C08802=1110.734,383.044,-89.612,-176.811,11.292,149.467
C08803=1110.731,383.291,-89.650,-176.808,11.295,149.467
C08804=1110.727,383.538,-89.689,-176.805,11.297,149.467
C08805=1110.724,383.785,-89.726,-176.802,11.300,149.467
C08806=1110.719,384.033,-89.763,-176.799,11.303,149.467
C08807=1110.716,384.280,-89.801,-176.796,11.306,149.467
C08808=1110.712,384.526,-89.839,-176.794,11.308,149.466
C08809=1110.709,384.774,-89.877,-176.791,11.310,149.466
C08810=1110.705,385.021,-89.915,-176.788,11.313,149.466
C08811=1110.702,385.268,-89.953,-176.785,11.316,149.466
C08812=1110.698,385.514,-89.990,-176.783,11.318,149.466
C08813=1110.694,385.762,-90.028,-176.780,11.321,149.466
C08814=1110.690,386.009,-90.066,-176.777,11.324,149.466
C08815=1110.687,386.256,-90.104,-176.774,11.327,149.466
C08816=1110.683,386.504,-90.142,-176.772,11.330,149.466
C08817=1110.680,386.750,-90.179,-176.769,11.332,149.466
C08818=1110.676,386.998,-90.218,-176.766,11.335,149.466
C08819=1110.672,387.244,-90.255,-176.763,11.337,149.466
C08820=1110.669,387.492,-90.293,-176.761,11.340,149.467
C08821=1110.665,387.739,-90.332,-176.758,11.343,149.467
C08822=1110.661,387.986,-90.369,-176.755,11.346,149.467
C08823=1110.658,388.233,-90.407,-176.753,11.349,149.467
C08824=1110.653,388.480,-90.446,-176.750,11.352,149.467
C08825=1110.650,388.727,-90.484,-176.747,11.355,149.467
C08826=1110.647,388.974,-90.522,-176.744,11.358,149.467
C08827=1110.643,389.221,-90.560,-176.742,11.361,149.467
C08828=1110.639,389.468,-90.598,-176.739,11.364,149.467
C08829=1110.636,389.715,-90.636,-176.737,11.367,149.467
C08830=1110.632,389.962,-90.674,-176.734,11.370,149.467
C08831=1110.629,390.209,-90.712,-176.731,11.374,149.467
C08832=1110.626,390.420,-90.745,-176.729,11.376,149.468
C08833=1110.622,390.632,-90.778,-176.726,11.379,149.468
C08834=1110.619,390.843,-90.810,-176.724,11.382,149.468
C08835=1110.616,391.055,-90.843,-176.722,11.385,149.468
C08836=1110.613,391.266,-90.876,-176.720,11.387,149.468
C08837=1110.610,391.477,-90.909,-176.717,11.390,149.468
C08838=1110.607,391.689,-90.941,-176.716,11.393,149.469
C08839=1110.603,391.900,-90.974,-176.713,11.396,149.469
C08840=1110.600,392.147,-91.012,-176.711,11.399,149.469
C08841=1110.596,392.395,-91.051,-176.707,11.403,149.469
C08842=1110.593,392.641,-91.089,-176.705,11.406,149.469
C08843=1110.589,392.888,-91.127,-176.702,11.409,149.470
C08844=1110.586,393.135,-91.165,-176.700,11.412,149.470
C08845=1110.582,393.382,-91.205,-176.697,11.416,149.470
C08846=1110.578,393.629,-91.242,-176.695,11.420,149.470
C08847=1110.574,393.876,-91.281,-176.692,11.423,149.471
C08848=1110.572,394.123,-91.319,-176.689,11.427,149.471
C08849=1110.567,394.370,-91.358,-176.687,11.430,149.471
C08850=1110.564,394.617,-91.396,-176.684,11.434,149.471
C08851=1110.560,394.864,-91.435,-176.682,11.438,149.472
C08852=1110.557,395.112,-91.473,-176.679,11.441,149.472
C08853=1110.553,395.358,-91.512,-176.676,11.445,149.472
C08854=1110.549,395.605,-91.550,-176.674,11.448,149.473
C08855=1110.546,395.852,-91.589,-176.671,11.453,149.473
C08856=1110.542,396.100,-91.627,-176.669,11.456,149.473
C08857=1110.539,396.346,-91.666,-176.666,11.460,149.474
C08858=1110.535,396.593,-91.704,-176.664,11.464,149.474
C08859=1110.531,396.840,-91.743,-176.661,11.468,149.474
C08860=1110.528,397.087,-91.782,-176.659,11.471,149.475
C08861=1110.524,397.334,-91.821,-176.656,11.476,149.475
C08862=1110.521,397.580,-91.859,-176.654,11.480,149.476
C08863=1110.517,397.828,-91.897,-176.651,11.483,149.476
C08864=1110.513,398.075,-91.937,-176.649,11.487,149.476
C08865=1110.510,398.321,-91.975,-176.646,11.492,149.477
C08866=1110.506,398.569,-92.014,-176.644,11.495,149.477
C08867=1110.503,398.816,-92.053,-176.642,11.500,149.478
C08868=1110.499,399.062,-92.091,-176.639,11.504,149.478
C08869=1110.495,399.310,-92.130,-176.637,11.508,149.479
C08870=1110.492,399.556,-92.169,-176.634,11.512,149.479
C08871=1110.488,399.803,-92.208,-176.632,11.516,149.480
C08872=1110.485,400.050,-92.247,-176.629,11.521,149.480
C08873=1110.481,400.298,-92.286,-176.627,11.525,149.481
C08874=1110.478,400.545,-92.325,-176.625,11.529,149.481
C08875=1110.474,400.791,-92.364,-176.622,11.533,149.482
C08876=1110.471,401.038,-92.402,-176.620,11.538,149.482
C08877=1110.467,401.285,-92.442,-176.617,11.542,149.483
C08878=1110.463,401.532,-92.480,-176.615,11.547,149.483
C08879=1110.459,401.779,-92.519,-176.612,11.551,149.484
C08880=1110.457,402.026,-92.558,-176.610,11.556,149.484
C08881=1110.453,402.273,-92.597,-176.608,11.560,149.485
C08882=1110.449,402.520,-92.637,-176.605,11.565,149.486
C08883=1110.446,402.767,-92.676,-176.603,11.570,149.486
C08884=1110.442,403.014,-92.715,-176.601,11.574,149.487
C08885=1110.438,403.261,-92.754,-176.599,11.579,149.488
C08886=1110.436,403.507,-92.793,-176.596,11.584,149.488
C08887=1110.431,403.753,-92.832,-176.594,11.588,149.489
C08888=1110.426,404.103,-92.887,-176.591,11.595,149.490
C08889=1110.422,404.451,-92.942,-176.588,11.602,149.491
C08890=1110.417,404.800,-92.998,-176.584,11.609,149.492
C08891=1110.411,405.148,-93.053,-176.581,11.616,149.493
C08892=1110.408,405.395,-93.093,-176.579,11.620,149.494
C08893=1110.404,405.642,-93.132,-176.576,11.626,149.494
C08894=1110.400,405.889,-93.171,-176.574,11.631,149.495
C08895=1110.398,406.135,-93.211,-176.572,11.636,149.496
C08896=1110.394,406.382,-93.250,-176.570,11.641,149.497
C08897=1110.391,406.629,-93.289,-176.568,11.646,149.497
C08898=1110.387,406.876,-93.328,-176.566,11.651,149.498
C08899=1110.383,407.123,-93.368,-176.563,11.657,149.499
C08900=1110.380,407.370,-93.407,-176.561,11.662,149.500
C08901=1110.376,407.616,-93.447,-176.559,11.667,149.501
C08902=1110.373,407.863,-93.486,-176.557,11.672,149.502
C08903=1110.369,408.110,-93.525,-176.555,11.678,149.503
C08904=1110.366,408.357,-93.565,-176.553,11.683,149.503
C08905=1110.362,408.604,-93.604,-176.551,11.688,149.504
C08906=1110.359,408.851,-93.644,-176.548,11.694,149.505
C08907=1110.356,409.098,-93.683,-176.546,11.699,149.506
C08908=1110.099,397.773,-91.950,-176.648,11.485,149.476
C08909=1110.102,397.527,-91.911,-176.651,11.480,149.475
C08910=1110.106,397.279,-91.873,-176.654,11.476,149.475
C08911=1110.109,397.032,-91.833,-176.656,11.473,149.474
C08912=1110.112,396.785,-91.795,-176.659,11.468,149.474
C08913=1110.117,396.539,-91.757,-176.661,11.465,149.474
C08914=1110.120,396.291,-91.719,-176.664,11.461,149.473
C08915=1110.123,396.044,-91.679,-176.667,11.457,149.473
C08916=1110.127,395.797,-91.641,-176.669,11.454,149.473
C08917=1110.131,395.551,-91.603,-176.672,11.449,149.472
C08918=1110.135,395.303,-91.564,-176.674,11.446,149.472
C08919=1110.138,395.057,-91.525,-176.677,11.442,149.472
C08920=1110.142,394.809,-91.487,-176.679,11.438,149.471
C08921=1110.145,394.563,-91.449,-176.682,11.434,149.471
C08922=1110.149,394.316,-91.410,-176.684,11.431,149.471
C08923=1110.153,394.069,-91.371,-176.687,11.428,149.470
C08924=1110.156,393.821,-91.333,-176.690,11.424,149.470
C08925=1110.160,393.574,-91.295,-176.692,11.420,149.470
C08926=1110.163,393.328,-91.256,-176.695,11.417,149.470
C08927=1110.167,393.080,-91.217,-176.698,11.413,149.469
C08928=1110.170,392.833,-91.180,-176.700,11.410,149.469
C08929=1110.175,392.587,-91.141,-176.703,11.406,149.469
C08930=1110.178,392.339,-91.103,-176.706,11.403,149.469
C08931=1110.182,392.092,-91.064,-176.708,11.400,149.469
C08932=1110.185,391.846,-91.026,-176.711,11.397,149.469
C08933=1110.191,391.437,-90.962,-176.715,11.391,149.468
C08934=1110.197,391.027,-90.900,-176.720,11.386,149.468
C08935=1110.203,390.618,-90.836,-176.724,11.380,149.468
C08936=1110.209,390.210,-90.773,-176.729,11.375,149.467
C08937=1110.212,389.962,-90.735,-176.731,11.372,149.467
C08938=1110.216,389.715,-90.696,-176.735,11.368,149.467
C08939=1110.220,389.468,-90.659,-176.737,11.365,149.467
C08940=1110.223,389.221,-90.621,-176.740,11.362,149.467
C08941=1110.227,388.975,-90.582,-176.743,11.359,149.467
C08942=1110.231,388.727,-90.544,-176.745,11.356,149.467
C08943=1110.234,388.480,-90.506,-176.748,11.353,149.467
C08944=1110.238,388.233,-90.468,-176.751,11.351,149.467
C08945=1110.242,387.986,-90.430,-176.754,11.347,149.466
C08946=1110.245,387.739,-90.392,-176.756,11.345,149.466
C08947=1110.249,387.492,-90.354,-176.759,11.341,149.466
C08948=1110.252,387.245,-90.316,-176.762,11.339,149.466
C08949=1110.256,386.998,-90.278,-176.765,11.336,149.466
C08950=1110.259,386.751,-90.240,-176.768,11.333,149.466
C08951=1110.264,386.504,-90.202,-176.771,11.330,149.466
C08952=1110.267,386.257,-90.164,-176.773,11.327,149.466
C08953=1110.270,386.009,-90.126,-176.775,11.325,149.466
C08954=1110.275,385.762,-90.088,-176.778,11.322,149.466
C08955=1110.278,385.515,-90.050,-176.781,11.319,149.466
C08956=1110.282,385.269,-90.013,-176.784,11.316,149.466
C08957=1110.285,385.021,-89.975,-176.787,11.314,149.466
C08958=1110.289,384.774,-89.938,-176.790,11.311,149.466
C08959=1110.293,384.527,-89.899,-176.792,11.309,149.466
C08960=1110.297,384.280,-89.862,-176.795,11.306,149.466
C08961=1110.300,384.033,-89.824,-176.798,11.304,149.466
C08962=1110.303,383.785,-89.786,-176.801,11.301,149.466
C08963=1110.307,383.539,-89.748,-176.803,11.299,149.467
C08964=1110.311,383.291,-89.710,-176.807,11.296,149.467
C08965=1110.315,383.044,-89.673,-176.810,11.293,149.467
C08966=1110.318,382.797,-89.635,-176.813,11.290,149.467
C08967=1110.322,382.550,-89.597,-176.817,11.288,149.467
C08968=1110.325,382.302,-89.560,-176.820,11.285,149.467
C08969=1110.329,382.056,-89.522,-176.823,11.282,149.467
C08970=1110.333,381.808,-89.484,-176.827,11.279,149.467
C08971=1110.337,381.562,-89.446,-176.830,11.276,149.467
C08972=1110.341,381.315,-89.410,-176.833,11.274,149.468
C08973=1110.344,381.067,-89.372,-176.836,11.271,149.468
C08974=1110.348,380.821,-89.334,-176.840,11.269,149.468
C08975=1110.352,380.573,-89.297,-176.843,11.266,149.468
C08976=1110.355,380.326,-89.259,-176.846,11.263,149.468
C08977=1110.359,380.078,-89.222,-176.850,11.260,149.468
C08978=1110.363,379.832,-89.184,-176.853,11.258,149.469
C08979=1110.366,379.584,-89.147,-176.856,11.255,149.469
C08980=1110.370,379.337,-89.110,-176.859,11.252,149.469
C08981=1110.374,379.091,-89.072,-176.863,11.250,149.469
C08982=1110.377,378.843,-89.035,-176.866,11.247,149.469
C08983=1110.381,378.596,-88.997,-176.870,11.244,149.469
C08984=1110.384,378.348,-88.960,-176.873,11.242,149.470
C08985=1110.389,378.137,-88.928,-176.875,11.240,149.470
C08986=1110.392,377.925,-88.896,-176.879,11.237,149.470
C08987=1110.394,377.714,-88.863,-176.881,11.235,149.470
C08988=1110.398,377.503,-88.832,-176.884,11.233,149.470
C08989=1110.401,377.291,-88.800,-176.887,11.231,149.470
C08990=1110.404,377.079,-88.768,-176.890,11.228,149.470
C08991=1110.407,376.868,-88.737,-176.892,11.226,149.471
C08992=1110.410,376.657,-88.705,-176.896,11.224,149.471
C08993=1110.414,376.410,-88.667,-176.899,11.221,149.471
C08994=1110.418,376.162,-88.630,-176.902,11.219,149.471
C08995=1110.422,375.915,-88.593,-176.906,11.216,149.471
C08996=1110.426,375.669,-88.556,-176.909,11.214,149.472
C08997=1110.429,375.421,-88.519,-176.912,11.212,149.472
C08998=1110.433,375.173,-88.482,-176.915,11.209,149.472
C08999=1110.437,374.926,-88.445,-176.919,11.207,149.472
C09000=1110.440,374.679,-88.407,-176.922,11.204,149.472
C09001=1110.444,374.432,-88.371,-176.925,11.202,149.473
C09002=1110.448,374.185,-88.334,-176.929,11.198,149.473
C09003=1110.451,373.937,-88.297,-176.933,11.196,149.473
C09004=1110.455,373.690,-88.259,-176.936,11.193,149.473
C09005=1110.459,373.443,-88.222,-176.939,11.191,149.473
C09006=1110.463,373.195,-88.185,-176.942,11.188,149.473
C09007=1110.466,372.948,-88.149,-176.946,11.186,149.474
C09008=1110.470,372.701,-88.112,-176.949,11.183,149.474
C09009=1110.474,372.454,-88.075,-176.952,11.181,149.474
C09010=1110.477,372.207,-88.037,-176.956,11.179,149.474
C09011=1110.481,371.960,-88.001,-176.959,11.176,149.475
C09012=1110.485,371.713,-87.964,-176.963,11.174,149.475
C09013=1110.489,371.466,-87.927,-176.966,11.171,149.475
C09014=1110.493,371.218,-87.890,-176.969,11.169,149.475
C09015=1110.496,370.971,-87.853,-176.973,11.166,149.476
C09016=1110.500,370.724,-87.817,-176.976,11.164,149.476
C09017=1110.504,370.476,-87.780,-176.979,11.161,149.476
C09018=1110.508,370.228,-87.743,-176.983,11.159,149.476
C09019=1110.511,369.982,-87.706,-176.986,11.157,149.477
C09020=1110.515,369.734,-87.669,-176.989,11.154,149.477
C09021=1110.519,369.487,-87.633,-176.993,11.152,149.477
C09022=1110.522,369.240,-87.596,-176.996,11.149,149.477
C09023=1110.526,368.992,-87.559,-176.999,11.147,149.477
C09024=1110.530,368.745,-87.522,-177.003,11.144,149.478
C09025=1110.534,368.498,-87.487,-177.006,11.142,149.478
C09026=1110.538,368.251,-87.450,-177.010,11.140,149.478
C09027=1110.541,368.004,-87.414,-177.013,11.137,149.478
C09028=1110.545,367.757,-87.377,-177.016,11.135,149.479
C09029=1110.549,367.509,-87.339,-177.020,11.132,149.479
C09030=1110.552,367.262,-87.303,-177.023,11.130,149.479
C09031=1110.557,367.014,-87.267,-177.027,11.128,149.479
C09032=1110.561,366.767,-87.230,-177.030,11.125,149.480
C09033=1110.564,366.520,-87.194,-177.033,11.123,149.480
C09034=1110.568,366.273,-87.157,-177.036,11.120,149.480
C09035=1110.571,366.026,-87.121,-177.040,11.118,149.480
C09036=1110.576,365.778,-87.085,-177.043,11.116,149.481
C09037=1110.579,365.530,-87.048,-177.047,11.113,149.481
C09038=1110.583,365.283,-87.011,-177.050,11.111,149.481
C09039=1110.586,365.036,-86.976,-177.053,11.108,149.481
C09040=1110.590,364.789,-86.939,-177.057,11.106,149.482
C09041=1110.594,364.577,-86.908,-177.060,11.104,149.482
C09042=1110.597,364.366,-86.877,-177.063,11.102,149.482
C09043=1110.600,364.154,-86.846,-177.065,11.100,149.482
C09044=1110.604,363.942,-86.814,-177.069,11.097,149.482
C09045=1110.607,363.731,-86.784,-177.071,11.096,149.483
C09046=1110.609,363.519,-86.752,-177.075,11.093,149.483
C09047=1110.613,363.307,-86.721,-177.077,11.092,149.483
C09048=1110.616,363.095,-86.691,-177.080,11.090,149.483
C09049=1110.620,362.848,-86.654,-177.083,11.087,149.484
C09050=1110.624,362.600,-86.618,-177.087,11.085,149.484
C09051=1110.628,362.353,-86.581,-177.090,11.083,149.484
C09052=1110.631,362.106,-86.546,-177.094,11.080,149.484
C09053=1110.635,361.859,-86.510,-177.097,11.078,149.485
C09054=1110.639,361.611,-86.474,-177.100,11.075,149.485
C09055=1110.642,361.364,-86.437,-177.103,11.073,149.485
C09056=1110.646,361.117,-86.402,-177.107,11.070,149.485
C09057=1110.650,360.869,-86.365,-177.110,11.068,149.486
C09058=1110.654,360.622,-86.329,-177.114,11.066,149.486
C09059=1110.658,360.375,-86.292,-177.117,11.063,149.486
C09060=1110.662,360.127,-86.257,-177.120,11.061,149.486
C09061=1110.665,359.880,-86.221,-177.124,11.059,149.487
C09062=1110.669,359.633,-86.185,-177.127,11.056,149.487
C09063=1110.673,359.385,-86.149,-177.131,11.054,149.487
C09064=1110.677,359.138,-86.113,-177.134,11.051,149.487
C09065=1110.680,358.891,-86.077,-177.137,11.049,149.488
C09066=1110.684,358.643,-86.041,-177.141,11.046,149.488
C09067=1110.688,358.395,-86.005,-177.144,11.044,149.488
C09068=1110.691,358.149,-85.969,-177.148,11.042,149.488
C09069=1110.695,357.901,-85.934,-177.151,11.039,149.489
C09070=1110.700,357.653,-85.898,-177.154,11.037,149.489
C09071=1110.703,357.406,-85.862,-177.158,11.034,149.489
C09072=1110.707,357.158,-85.826,-177.161,11.032,149.489
C09073=1110.710,356.911,-85.790,-177.165,11.030,149.490
C09074=1110.715,356.664,-85.754,-177.168,11.027,149.490
C09075=1110.719,356.417,-85.719,-177.171,11.025,149.490
C09076=1110.723,356.169,-85.683,-177.174,11.022,149.490
C09077=1110.726,355.922,-85.648,-177.178,11.020,149.491
C09078=1110.730,355.674,-85.612,-177.181,11.018,149.491
C09079=1110.734,355.427,-85.577,-177.185,11.015,149.491
C09080=1110.738,355.180,-85.540,-177.188,11.013,149.491
C09081=1110.741,354.932,-85.504,-177.191,11.010,149.492
C09082=1110.745,354.685,-85.469,-177.195,11.008,149.492
C09083=1110.749,354.437,-85.433,-177.198,11.006,149.492
C09084=1110.753,354.190,-85.398,-177.201,11.003,149.492
C09085=1110.757,353.943,-85.362,-177.205,11.001,149.493
C09086=1110.760,353.695,-85.327,-177.208,10.998,149.493
C09087=1110.765,353.447,-85.291,-177.211,10.996,149.493
C09088=1110.768,353.200,-85.255,-177.215,10.993,149.493
C09089=1110.772,352.952,-85.220,-177.218,10.991,149.493
C09090=1110.776,352.706,-85.184,-177.221,10.988,149.494
C09091=1110.780,352.458,-85.149,-177.225,10.986,149.494
C09092=1110.784,352.211,-85.113,-177.228,10.984,149.494
C09093=1110.788,351.962,-85.079,-177.231,10.981,149.495
C09094=1110.791,351.715,-85.043,-177.235,10.979,149.495
C09095=1110.795,351.467,-85.007,-177.238,10.976,149.495
C09096=1110.799,351.221,-84.972,-177.241,10.974,149.495
C09097=1110.802,351.009,-84.942,-177.244,10.972,149.495
C09098=1110.806,350.796,-84.912,-177.246,10.970,149.496
C09099=1110.809,350.585,-84.881,-177.250,10.968,149.496
C09100=1110.812,350.373,-84.851,-177.252,10.966,149.496
C09101=1110.815,350.161,-84.820,-177.255,10.963,149.496
C09102=1110.819,349.950,-84.791,-177.258,10.962,149.496
C09103=1110.822,349.738,-84.761,-177.261,10.959,149.496
C09104=1110.825,349.527,-84.730,-177.264,10.957,149.497
C09105=1110.829,349.278,-84.695,-177.267,10.955,149.497
C09106=1110.833,349.031,-84.660,-177.270,10.952,149.497
C09107=1110.837,348.784,-84.625,-177.273,10.950,149.497
C09108=1110.841,348.536,-84.590,-177.277,10.947,149.498
C09109=1110.845,348.288,-84.554,-177.280,10.944,149.498
C09110=1110.848,348.041,-84.519,-177.282,10.943,149.498
C09111=1110.853,347.794,-84.484,-177.286,10.940,149.498
C09112=1110.856,347.546,-84.449,-177.289,10.938,149.498
C09113=1110.860,347.299,-84.413,-177.292,10.935,149.498
C09114=1110.865,347.051,-84.379,-177.296,10.933,149.499
